// TwinCAT 3 PLC project MONETcommon
// Title: MONETcommon
// Company: IAG
// ProjectVersion: 0.5.0
// ProgramVersion: 3.1.4024.0
// libraries:
//   AstroBROT, * (BROT)
//   BROTLib, * (BROT)
//   HalfBROT, * (BROT)
//   Tc2_MC2, * (Beckhoff Automation GmbH)
//   Tc2_Standard, * (Beckhoff Automation GmbH)
//   Tc2_System, * (Beckhoff Automation GmbH)
//   Tc2_Utilities, * (Beckhoff Automation GmbH)
// project tree:
//   / E_ModeLanguage.TcDUT, FB_MonetCabinetControl.TcPOU, FB_MonetCoverControl.TcPOU, FB_MonetDiagnostics.TcPOU, FB_MonetMqttWatchdog.TcPOU, FB_MonetPendantControl.TcPOU, FB_MonetPowerMonitoring.TcPOU, FB_MonetSafetyHandling.TcPOU, F_AzimuthOffsetOnAxis.TcPOU, FB_MonetTelescopeControl.TcPOU, Global_Version.TcGVL

// ---- E_ModeLanguage.TcDUT
TYPE E_ModeLanguage :(Deutsch:=1,English:=2);


END_TYPE

// ---- Global_Version.TcGVL
{attribute 'qualified_only'}
VAR_GLOBAL CONSTANT
	// Mirrors Beckhoff's own Global_Version.stLibVersion_* pattern (see ST_LibVersion),
	// which only covers Tc2_*/Tc3_* library references, not custom ones -- until now: this
	// GVL uses Beckhoff's own naming exactly, so it merges into a consumer's Global_Version.
	// Kept in sync with <ProjectVersion> in MONETcommon.plcproj at release time.
	stLibVersion_MONETcommon : ST_LibVersion := (
		iMajor := 0,
		iMinor := 5,
		iBuild := 0,
		iRevision := 0,
		nFlags := 1,
		sVersion := '0.5.0'
	);
END_VAR

// ---- FB_MonetCabinetControl.TcPOU
FUNCTION_BLOCK FB_MonetCabinetControl
VAR_INPUT
END_VAR
VAR_OUTPUT
	bCabinetOverTemp	: BOOL;	// cabinet temperature (BT1) is critical (>60°C); not wired to any stop/park action yet, see MONETcommon#21
END_VAR
VAR
	// AT%I*/AT%Q* below are mapped directly on this FB: only one instance per PLC is
	// supported, a second instance would collide on the same physical hardware.
	inKeyLocal			AT%I*: BOOL;	//DIN3 0.2
	inButtonStart		AT%I*: BOOL;	//DIN4 0.3
	inButtonStop		AT%I*: BOOL;	//DIN5 0.4
	inButtonReset		AT%I*: BOOL;	//DIN8 0.7
	inCabinetTemp		AT%I*: INT;		//BT1	
	inKeyClearBrakes	AT%I*: BOOL;	//DIN15 1.6
	outLampPower		AT%Q*: BOOL;	//DOUT1 0.0
	outLampManual		AT%Q*: BOOL;	//DOUT2 0.1
	outLampError		AT%Q*: BOOL;	//DOUT3 0.2	
	cabinetTemp				: REAL;
	tempWarning				: SR;
	tempCritical			: SR;
	tempEvent				: FB_EventLog;
	tempCriticalEvent		: FB_EventLog;
	blinkErrorLamp			: FB_BLINK;
	blinkPowerLamp			: FB_BLINK;
	commTimer 				: TON := (PT:=T#5S);
	fbComm					: I_Comm;
END_VAR

// check temperature
cabinetTemp := INT_TO_REAL(inCabinetTemp) / 10.0;
tempWarning(SET1 := cabinetTemp > 50.0, RESET := cabinetTemp < 40.0);
tempCritical(SET1 := cabinetTemp > 60.0, RESET := cabinetTemp < 50.0);
bCabinetOverTemp := tempCritical.Q1;

// blinking lights
blinkErrorLamp(Q => outLampError);
blinkPowerLamp(Q => outLampPower);

// telemetry
commTimer(IN:=TRUE);
IF commTimer.Q THEN
	commTimer(IN:=FALSE);
	fbComm.Publish('electronics', 'base', 'MainCabinetTemperature', LREAL_TO_FMTSTR(cabinetTemp, 2, TRUE));
END_IF

// events
tempEvent(	
	Trigger 		:= tempWarning.Q1, 
	Level 			:= ADSLOG_MSGTYPE_WARN,
	FormatString 	:= 'Main cabinet temperature warning:	%s',
	OnMessage 		:= LREAL_TO_FMTSTR(cabinetTemp, 1, TRUE),
	comm			:= fbComm);
tempCriticalEvent(	
	Trigger 		:= tempCritical.Q1, 
	Level 			:= ADSLOG_MSGTYPE_ERROR,
	FormatString 	:= 'Main cabinet temperature is critical:	%s!',
	OnMessage 		:= LREAL_TO_FMTSTR(cabinetTemp, 1, TRUE),
	comm			:= fbComm);

// deprecated: kept for existing callers (MONETN, MONETS MAIN), use AreBrakesCleared instead
METHOD PUBLIC AreBreakesCleared : BOOL
VAR_INPUT
END_VAR
AreBreakesCleared := THIS^.AreBrakesCleared();
END_METHOD

METHOD PUBLIC AreBrakesCleared : BOOL
VAR_INPUT
END_VAR
AreBrakesCleared := inKeyClearBrakes;
END_METHOD

//FB_Init is always available implicitly and it is used primarily for initialization.
//The return value is not evaluated. For a specific influence, you can also declare the
//methods explicitly and provide additional code there with the standard initialization
//code. You can evaluate the return value.
METHOD FB_Init: BOOL
VAR_INPUT
    bInitRetains	: BOOL; // TRUE: the retain variables are initialized (reset warm / reset cold)
    bInCopyCode		: BOOL;  // TRUE: the instance will be copied to the copy code afterward (online change)
	comm			: I_Comm;	   
END_VAR
THIS^.fbComm := comm;
END_METHOD

METHOD PUBLIC IsResetPushed : BOOL
VAR_INPUT
END_VAR
IsResetPushed := inButtonReset;
END_METHOD

METHOD PUBLIC IsStartPushed : BOOL
VAR_INPUT
END_VAR
IsStartPushed := inButtonStart;
END_METHOD

METHOD PUBLIC IsStopPushed : BOOL
VAR_INPUT
END_VAR
IsStopPushed := NOT inButtonStop;
END_METHOD

PROPERTY KeyLocal : BOOL
GET
KeyLocal := inKeyLocal;
END_GET
END_PROPERTY

METHOD PUBLIC SetBlinkError : BOOL
VAR_INPUT
	mode	: E_Blink;
END_VAR
blinkErrorLamp.blink := mode;
END_METHOD

METHOD PUBLIC SetBlinkPower : BOOL
VAR_INPUT
	mode	: E_Blink;
END_VAR
blinkPowerLamp.blink := mode;
END_METHOD

METHOD PUBLIC SetManualLamp : BOOL
VAR_INPUT
	enable	: BOOL;
END_VAR
outLampManual := enable;
END_METHOD

END_FUNCTION_BLOCK

// ---- FB_MonetCoverControl.TcPOU
FUNCTION_BLOCK FB_MonetCoverControl IMPLEMENTS I_MirrorCovers
VAR_INPUT
	bReset				: BOOL;		// resets all drives after an error has occurred
	// M3: bOpen/bClose are also written internally (cleared on completion) and are meant
	// to be driven only via the Open()/Close() methods, not wired externally every scan
	// (consumers currently call CoverControl() with no parameters).
	bOpen				: BOOL;		// open the cover in proper order
	bClose				: BOOL;		// close the cover in proper order
	
	// telemetry interval
	fTelemetryInterval		: TIME := T#5S;	
END_VAR
VAR_OUTPUT
	bAllOpen			: BOOL;		// all covers are open
	bAllClosed			: BOOL;		// all covers are closed
	bError				: BOOL;		// any cover-driver reports an error
END_VAR
VAR
	fbComm				: I_Comm;
	tonComm 			: TON := (PT:=fTelemetryInterval);	

	// AT%I*/AT%Q* below are mapped directly on this FB: only one instance per PLC is
	// supported, a second instance would collide on the same physical hardware.
	// output signals for opening/closing covers
	OabOpenCover  AT%Q* : ARRAY[1..3] OF BOOL;	// open cover1-3 command
	OabCloseCover AT%Q* : ARRAY[1..3] OF BOOL;   // close cover1-3 command
	
	// limit switches
	IabCoverOpen	AT%I* : ARRAY[1..3] OF BOOL;	// limit coper 1 open switch
	IabCoverClosed	AT%I* : ARRAY[1..3] OF BOOL;	// limit coper 1 closed switch
	
	// status
	abCoverOpen			: ARRAY[1..3] OF BOOL;	// cover is open
	abCoverClosed		: ARRAY[1..3] OF BOOL;	// cover is closed
	abCoverError			: ARRAY[1..3] OF BOOL;	// cover has error
	afbCoverEvent			: ARRAY[1..3] OF FB_EventLog;	// cover event
	afbTimeoutEvent : ARRAY[1..3] OF FB_EventLog;	// cover has timeout

	// M3: drive timeout if a cover does not reach its target limit switch within PT;
	// TUNE PT to the actual drive on site, 60s is an untested placeholder.
	atonMoveTimeout		: ARRAY[1..3] OF TON;
	asrCoverTimeout		: ARRAY[1..3] OF SR;	// latched until bReset, see the TON note above
	abCoverTimeout		: ARRAY[1..3] OF BOOL;
	
	srErrorTrigger			: SR;	// trigger for error
	
	fbCoversOpenedEvent		: FB_EventLog; // log if covers are open
	fbCoversClosedEvent		: FB_EventLog; // log if covers are closed
	fbCoversErrorEvent		: FB_EventLog; // Event log for a generic drive error
	
	i	: UINT;
END_VAR

(*
This is the control for the two (three) telescope covers. 
The correct order for opening is 1->3->2 and for closing 2->3->1.
GVL Open and close signals are inverted
*)

// close has precedence over open
IF bClose THEN
	bOpen := FALSE;
END_IF

// do stuff for all covers
FOR i := 1 TO 3 BY 1 DO
	// limit switches are inverted
    abCoverOpen[i]   := NOT IabCoverOpen[i];
	abCoverClosed[i] := NOT IabCoverClosed[i];

	// errors occur if covers are both opened and closed
	abCoverError[i] := abCoverOpen[i] AND abCoverClosed[i];

	// M3: a cover being driven but not reaching its target switch is also an error,
	// and must stop driving the output (gated below), not just log and keep pushing.
	atonMoveTimeout[i](IN := OabOpenCover[i] OR OabCloseCover[i], PT := T#60S);
	asrCoverTimeout[i](SET1 := atonMoveTimeout[i].Q, RESET := bReset, Q1 => abCoverTimeout[i]);
	abCoverError[i] := abCoverError[i] OR abCoverTimeout[i];
END_FOR;

// close 2->3->1
OabCloseCover[2] := bClose AND NOT abCoverClosed[2] AND NOT abCoverTimeout[2];
OabCloseCover[3] := bClose AND NOT abCoverClosed[3] AND abCoverClosed[2] AND NOT abCoverTimeout[3];
OabCloseCover[1] := bClose AND NOT abCoverClosed[1] AND abCoverClosed[2] AND abCoverClosed[3] AND NOT abCoverTimeout[1];

// open 1->3->2
OabOpenCover[1] := bOpen AND NOT abCoverOpen[1] AND NOT abCoverTimeout[1];
OabOpenCover[3] := bOpen AND NOT abCoverOpen[3] AND abCoverOpen[1] AND NOT abCoverTimeout[3];
OabOpenCover[2] := bOpen AND NOT abCoverOpen[2] AND abCoverOpen[1] AND abCoverOpen[3] AND NOT abCoverTimeout[2];

// we are open, if all covers are open
bAllOpen := abCoverOpen[1] AND abCoverOpen[2] AND abCoverOpen[3];
// we are closed, if all covers are closed
bAllClosed := abCoverClosed[1] AND abCoverClosed[2] AND abCoverClosed[3];

// error indicates an axis error on any axis
srErrorTrigger(
	SET1 := abCoverError[1] OR abCoverError[2] OR abCoverError[3],
	RESET := bReset,
	Q1 => bError);

// clear reset, if no error present
IF NOT bError THEN
	bReset := FALSE;
END_IF

IF bAllClosed THEN
	bClose := FALSE;
END_IF

IF bAllOpen THEN
	bOpen := FALSE;
END_IF

fbCoversErrorEvent.OnMessage := 'Cover drive error';
IF bError THEN
	IF abCoverError[3] THEN 
		fbCoversErrorEvent.OnMessage := 'Cover 3 has a drive error.';
	END_IF
	IF abCoverError[2] THEN 
		fbCoversErrorEvent.OnMessage := 'Cover 2 has a drive error.';
	END_IF
	IF abCoverError[1] THEN 
		fbCoversErrorEvent.OnMessage := 'Cover 1 has a drive error.';
	END_IF
END_IF

// send telemetry
tonComm.PT := fTelemetryInterval;	// M3: fTelemetryInterval was only applied at init otherwise
tonComm(IN:=TRUE);
IF tonComm.Q THEN // publish new payload every second
	tonComm(IN:=FALSE);
	THIS^._SendTelemetry();	
END_IF

fbCoversErrorEvent(
	Trigger 	:= bError, 
   	Level   	:= ADSLOG_MSGTYPE_ERROR, 
	comm 		:= fbComm);

// raise an error, if both opened and closed signals are activated
// handle RoboTel differently
afbCoverEvent[1](
	Trigger   	:= abCoverOpen[1] AND abCoverClosed[1],
	Level     	:= ADSLOG_MSGTYPE_ERROR, 
	OnMessage 	:= 'Cover1: limit switch error', 
	comm	 	:= fbComm);

afbCoverEvent[2](
	Trigger   	:= abCoverOpen[2] AND abCoverClosed[2],
    Level     	:= ADSLOG_MSGTYPE_ERROR, 
	OnMessage 	:= 'Cover2: limit switch error', 
	comm      	:= fbComm);

afbCoverEvent[3](
	Trigger   	:= abCoverOpen[3] AND abCoverClosed[3],
	Level     	:= ADSLOG_MSGTYPE_ERROR, 
	OnMessage 	:= 'Cover3: limit switch error', 
	comm 	  	:= fbComm);

//trigger an event, if we encounter a timeout
afbTimeoutEvent[1](
	Trigger   	:= abCoverTimeout[1],
	Level     	:= ADSLOG_MSGTYPE_ERROR,
	OnMessage 	:= 'Cover1: Timeout',
	comm 		:= fbComm);
afbTimeoutEvent[2](
	Trigger   	:= abCoverTimeout[2],
 	Level     	:= ADSLOG_MSGTYPE_ERROR,
	OnMessage 	:= 'Cover2: Timeout',
	comm 		:= fbComm);
afbTimeoutEvent[3](
	Trigger   	:= abCoverTimeout[3],
	Level     	:= ADSLOG_MSGTYPE_ERROR,
	OnMessage 	:= 'Cover3: Timeout',
	comm 		:= fbComm);

// Log if we are opened
fbCoversOpenedEvent(
	Trigger   	:= bAllOpen,
	Level     	:= ADSLOG_MSGTYPE_WARN,
	OnMessage 	:= 'All covers are open',
	comm 		:= fbComm);
	
//log if we are closed
fbCoversClosedEvent(
	Trigger   	:= bAllClosed,
	Level     	:= ADSLOG_MSGTYPE_HINT,
	OnMessage 	:= 'All covers are closed',
	comm 		:= fbComm);

METHOD _SendTelemetry : BOOL
VAR_INPUT
END_VAR
IF bAllClosed THEN
	fbComm.Publish('telescope', 'dome', 'AUXILIARY.COVER.REALPOS', '0.0');
ELSIF bAllOpen THEN
	fbComm.Publish('telescope', 'dome', 'AUXILIARY.COVER.REALPOS', '1.0');
ELSE
	fbComm.Publish('telescope', 'dome', 'AUXILIARY.COVER.REALPOS', '0.5');
END_IF
END_METHOD

METHOD Close : BOOL
VAR_INPUT
END_VAR
bOpen := FALSE;
bClose := TRUE;
END_METHOD

PROPERTY Closed : BOOL
GET
Closed := bAllClosed;
END_GET
END_PROPERTY

PROPERTY Error : BOOL
GET
Error := bError;
END_GET
END_PROPERTY

//FB_Init is always available implicitly and it is used primarily for initialization.
//The return value is not evaluated. For a specific influence, you can also declare the
//methods explicitly and provide additional code there with the standard initialization
//code. You can evaluate the return value.
METHOD FB_Init: BOOL
VAR_INPUT
    bInitRetains	: BOOL; // TRUE: the retain variables are initialized (reset warm / reset cold)
    bInCopyCode		: BOOL;  // TRUE: the instance will be copied to the copy code afterward (online change)
	comm			: I_Comm;   
END_VAR
THIS^.fbComm := comm;
END_METHOD

METHOD Open : BOOL
VAR_INPUT
END_VAR
bOpen := TRUE;
bClose := FALSE;
END_METHOD

PROPERTY Opened : BOOL
GET
Opened := bAllOpen;
END_GET
END_PROPERTY

METHOD Reset : BOOL
VAR_INPUT
END_VAR
bReset := TRUE;
Reset := TRUE;
END_METHOD

END_FUNCTION_BLOCK

// ---- FB_MonetDiagnostics.TcPOU
// Diagnostics telemetry (measurement 'diagnostics', location 'base'): telescope interrupted/ready/busy/stopped,
// per-axis error, error ID and enable, safety error/estop/state. Each value is published when it changes, plus a full
// snapshot every tHeartbeat so a human scanning history can tell the system was actively reporting, not just silent.
// Booleans are retained by the broker (FB_Comm_MQTT_Influx.Publish). Moved unchanged from MONETS's MAIN so that
// MONET/S and MONET/N share it (IAG specs/plans/2026-09-09-extended-diagnostics-telemetry-proposal.md).
FUNCTION_BLOCK FB_MonetDiagnostics
VAR_INPUT
	fbTelescope		: REFERENCE TO FB_MonetTelescopeControl;
	fbElevation		: REFERENCE TO FB_ElevationControl;
	fbAzimuth		: REFERENCE TO FB_AzimuthControl;
	fbDerotator		: REFERENCE TO FB_DerotatorControl;
	fbFocus			: REFERENCE TO FB_FocusControl;
	fbSafety		: REFERENCE TO FB_MonetSafetyHandling;
	tHeartbeat		: TIME := T#30S;	// republish the full snapshot on this cadence even with no change
END_VAR
VAR
	fbComm					: I_Comm;
	tonHeartbeat			: TON;
	bHeartbeatTick			: BOOL;
	bLastInterrupted		: BOOL;
	bLastElevationError		: BOOL;
	bLastAzimuthError		: BOOL;
	bLastDerotatorError		: BOOL;
	bLastFocusError			: BOOL;
	bLastElevationEnabled	: BOOL;
	bLastAzimuthEnabled		: BOOL;
	bLastDerotatorEnabled	: BOOL;
	bLastSafetyError		: BOOL;
	bLastSafetyEstop		: BOOL;
	bLastSafetyState		: BOOL;
	bLastTelescopeReady		: BOOL;
	bLastTelescopeBusy		: BOOL;
	bLastTelescopeStopped	: BOOL;
END_VAR

IF NOT (__ISVALIDREF(fbTelescope) AND __ISVALIDREF(fbElevation) AND __ISVALIDREF(fbAzimuth) AND
	__ISVALIDREF(fbDerotator) AND __ISVALIDREF(fbFocus) AND __ISVALIDREF(fbSafety)) THEN
	RETURN;
END_IF

tonHeartbeat(IN := TRUE, PT := tHeartbeat);
bHeartbeatTick := tonHeartbeat.Q;
IF bHeartbeatTick THEN
	tonHeartbeat(IN := FALSE);
END_IF

IF (fbTelescope.bInterrupted <> bLastInterrupted) OR bHeartbeatTick THEN
	fbComm.Publish('diagnostics', 'base', 'Interrupted', BOOL_TO_STRING(fbTelescope.bInterrupted));
	bLastInterrupted := fbTelescope.bInterrupted;
END_IF

IF (fbElevation.bError <> bLastElevationError) OR bHeartbeatTick THEN
	fbComm.Publish('diagnostics', 'base', 'ElevationError', BOOL_TO_STRING(fbElevation.bError));
	fbComm.Publish('diagnostics', 'base', 'ElevationErrorID', UDINT_TO_STRING(fbElevation.nErrorID));
	bLastElevationError := fbElevation.bError;
END_IF
IF (fbAzimuth.bError <> bLastAzimuthError) OR bHeartbeatTick THEN
	fbComm.Publish('diagnostics', 'base', 'AzimuthError', BOOL_TO_STRING(fbAzimuth.bError));
	fbComm.Publish('diagnostics', 'base', 'AzimuthErrorID', UDINT_TO_STRING(fbAzimuth.nErrorID));
	bLastAzimuthError := fbAzimuth.bError;
END_IF
IF (fbDerotator.bError <> bLastDerotatorError) OR bHeartbeatTick THEN
	fbComm.Publish('diagnostics', 'base', 'DerotatorError', BOOL_TO_STRING(fbDerotator.bError));
	fbComm.Publish('diagnostics', 'base', 'DerotatorErrorID', UDINT_TO_STRING(fbDerotator.nErrorID));
	bLastDerotatorError := fbDerotator.bError;
END_IF
IF (fbFocus.bError <> bLastFocusError) OR bHeartbeatTick THEN
	fbComm.Publish('diagnostics', 'base', 'FocusError', BOOL_TO_STRING(fbFocus.bError));
	fbComm.Publish('diagnostics', 'base', 'FocusErrorID', UDINT_TO_STRING(fbFocus.nErrorID));
	bLastFocusError := fbFocus.bError;
END_IF

IF (fbElevation.bEnable <> bLastElevationEnabled) OR bHeartbeatTick THEN
	fbComm.Publish('diagnostics', 'base', 'ElevationEnabled', BOOL_TO_STRING(fbElevation.bEnable));
	bLastElevationEnabled := fbElevation.bEnable;
END_IF
IF (fbAzimuth.bEnable <> bLastAzimuthEnabled) OR bHeartbeatTick THEN
	fbComm.Publish('diagnostics', 'base', 'AzimuthEnabled', BOOL_TO_STRING(fbAzimuth.bEnable));
	bLastAzimuthEnabled := fbAzimuth.bEnable;
END_IF
IF (fbDerotator.bEnable <> bLastDerotatorEnabled) OR bHeartbeatTick THEN
	fbComm.Publish('diagnostics', 'base', 'DerotatorEnabled', BOOL_TO_STRING(fbDerotator.bEnable));
	bLastDerotatorEnabled := fbDerotator.bEnable;
END_IF

IF (fbSafety.error <> bLastSafetyError) OR bHeartbeatTick THEN
	fbComm.Publish('diagnostics', 'base', 'SafetyError', BOOL_TO_STRING(fbSafety.error));
	bLastSafetyError := fbSafety.error;
END_IF
IF (fbSafety.estop <> bLastSafetyEstop) OR bHeartbeatTick THEN
	fbComm.Publish('diagnostics', 'base', 'SafetyEstop', BOOL_TO_STRING(fbSafety.estop));
	bLastSafetyEstop := fbSafety.estop;
END_IF
IF (fbSafety.state <> bLastSafetyState) OR bHeartbeatTick THEN
	fbComm.Publish('diagnostics', 'base', 'SafetyState', BOOL_TO_STRING(fbSafety.state));
	bLastSafetyState := fbSafety.state;
END_IF

IF (fbTelescope.bReady <> bLastTelescopeReady) OR bHeartbeatTick THEN
	fbComm.Publish('diagnostics', 'base', 'TelescopeReady', BOOL_TO_STRING(fbTelescope.bReady));
	bLastTelescopeReady := fbTelescope.bReady;
END_IF
IF (fbTelescope.bBusy <> bLastTelescopeBusy) OR bHeartbeatTick THEN
	fbComm.Publish('diagnostics', 'base', 'TelescopeBusy', BOOL_TO_STRING(fbTelescope.bBusy));
	bLastTelescopeBusy := fbTelescope.bBusy;
END_IF
IF (fbTelescope.bStopped <> bLastTelescopeStopped) OR bHeartbeatTick THEN
	fbComm.Publish('diagnostics', 'base', 'TelescopeStopped', BOOL_TO_STRING(fbTelescope.bStopped));
	bLastTelescopeStopped := fbTelescope.bStopped;
END_IF

METHOD FB_Init: BOOL
VAR_INPUT
    bInitRetains	: BOOL; // TRUE: the retain variables are initialized (reset warm / reset cold)
    bInCopyCode		: BOOL;  // TRUE: the instance will be copied to the copy code afterward (online change)
	comm			: I_Comm;
END_VAR
THIS^.fbComm := comm;
END_METHOD

END_FUNCTION_BLOCK

// ---- FB_MonetTelescopeControl.TcPOU
FUNCTION_BLOCK FB_MonetTelescopeControl EXTENDS FB_AltAzTelescopeControl IMPLEMENTS I_AltAzTelescope
VAR_INPUT
	fbFocus				: I_Focus;
	fbCovers			: I_MirrorCovers;
	fbBrake				: I_Brake;	
	fbHydraulics   		: I_Hydraulics;
	fbElevation			: REFERENCE TO FB_ElevationControl;
	fbAzimuth			: REFERENCE TO FB_AzimuthControl;
	fbDerotator			: REFERENCE TO FB_DerotatorControl;

	fbPointing			: REFERENCE TO FB_PointingModelForward;
	fbPointingInverse	: REFERENCE TO FB_PointingModelInversion;

	bBrakeClearing		: BOOL	:= TRUE;

	// M6: applied to every commanded elevation move (Goto/Home/Park/PowerOn/Slew, not
	// the computed tracking rate), NOT just _HomeTelescope despite the old name.
	// 5.0 deg/s confirmed correct on-site for MONETS; 10.0 was too fast.
	fElevationMoveVelocity : LREAL := 5.0;
END_VAR
VAR_OUTPUT
	fDerotatorSign		: LREAL := 1.0;	// derotator
	
	fElevationPointingOffset : LREAL;
	fAzimuthPointingOffset : LREAL;
	fElevationPointingOffset2 : LREAL;
	fAzimuthPointingOffset2 : LREAL;
	
	fRightAscensionCurrentSky: LREAL;
	fDeclinationCurrentSky: LREAL;

	fDerotatorVelocity	: LREAL;	// rotational velocity of the derotator
	fElevationVelocity	: LREAL;	// rotational velocity of the elevation
	fAzimuthVelocity	: LREAL;	// rotational velocity of the elevation
END_VAR
VAR
	// M1: internal (non-axis) errors from the Goto/Home/Slew state machines, latched
	// until bReset since bError/nErrorID are otherwise recomputed from the axes every
	// scan and would silently wipe these within the same cycle they're set in.
	bSoftwareError		: BOOL;
	nSoftwareErrorID	: UINT;
	SoftwareErrorEvent	: FB_EventLog;

	// #26 / ADR 0001 option 1: auto-clear a latched bInterrupted if nothing has been
	// requested for a while, since the normal arbitration path can never do it on its
	// own (bReady needs the axes enabled, axis enable needs bInterrupted already clear).
	// Visible, not silent: logged and counted, not just quietly cleared.
	bInterruptedIdle			: BOOL;
	tonInterruptedAutoClear		: TON;
	InterruptedAutoClearEvent	: FB_EventLog;
END_VAR
VAR PERSISTENT
	nInterruptedAutoClearCount	: UDINT;	// how many times auto-clear has fired, ever
END_VAR

// revert fDut1 (set via the Dut1 property, e.g. from an external time bridge over MQTT) to its
// safe 0.0 default if nothing fresh arrives for a while, instead of serving an arbitrarily
// stale UT1-UTC correction forever. FB_AltAzTelescopeControl's own body is never called (this FB
// doesn't call SUPER^() in its main body), so this has to live here rather than up there.
tonDut1Stale(IN := NOT bDut1Received, PT := T#10M);
bDut1Received := FALSE;
IF tonDut1Stale.Q THEN
	fDut1 := 0.0;
END_IF

// get the system time; fJd only follows the clock while the clock is valid (synced, see FB_AstroClock)
fbTime();
IF fbTime.bValid THEN
	fJd := DateTime2JD(fbTime.time_RTCEX2);
END_IF
fLst := CT2LST(telescopeConfig.longitude, fJd);

// without a trustworthy time nothing may be pointed or tracked: refuse through the normal stop path
IF NOT fbTime.bValid AND (bGoto OR bSlew OR bTrack) THEN
	bStop := TRUE;
END_IF

// set reset state either by hardware (key pressed) or by software (set by e.g. tcs)
rtrigReset(CLK := bReset);

IF bReset THEN
	bHorizonError := FALSE; // if reset, the bHorizonError can be switched off
	bSoftwareError := FALSE;
	
	// reset the stages of all statemachine methods
	bInterrupted := TRUE; 
	_HomeTelescope();
	_GotoTelescope();
	_SlewTelescope();
	_ParkTelescope();
	bInterrupted := FALSE;
END_IF

// get error ID, reset if bReset command is set
IF fbAzimuth.Error THEN
	nErrorID := fbAzimuth.nErrorID;
	IF bReset THEN
		fbAzimuth.Reset();
	END_IF
ELSIF fbElevation.bError THEN
	nErrorID := fbElevation.nErrorID;
	IF bReset THEN
		fbElevation.Reset();
	END_IF
ELSIF fbDerotator.bError THEN
	nErrorID := fbDerotator.nErrorID;
	IF bReset THEN
		fbDerotator.Reset();
	END_IF	
ELSIF fbFocus.Error THEN
	nErrorID := fbFocus.ErrorID;
	IF bReset THEN
		fbFocus.Reset();
	END_IF
ELSIF bSoftwareError THEN
	nErrorID := nSoftwareErrorID;
END_IF

// fSlewTime
fSlewTime :=  MAX(MAX(fbElevation.fSlewTime, fbAzimuth.fSlewTime), fbDerotator.fSlewTime);

bError := fbElevation.Error OR
		 fbAzimuth.bError OR
		 fbFocus.Error OR
		 fbDerotator.bError OR
		 bSoftwareError;
			
IF bError THEN
	bTrack := 	FALSE;
	bGoto := 	FALSE;
	bSlew := 	FALSE;
	fbElevation.Enable := FALSE;
	fbAzimuth.Enable := FALSE;
	fbDerotator.Enable := FALSE;
ELSE
	nErrorID := 0;
END_IF

IF fbElevation.bError THEN
	fbElevation.Enable := FALSE;
	fbAzimuth.Enable := FALSE;
	fbDerotator.Enable := FALSE;
	fbBrake.CloseBrake();
END_IF

eq2hor(
	ra := fRightAscension,
	dec := fDeclination,
	lon := telescopeConfig.longitude,
	lat := telescopeConfig.latitude,
	altitude := telescopeConfig.altitude,
	JD := fJd + fTimeOffset,
	dut1 := fDut1,
	refract_to_observed := TRUE,
	// refract := FALSE,
	alt => fElevationCalc,
	az => fAzimuthCalc,
	ha => fHourAngleCalc);

// apply pointing model
fbPointing(
	fAzimuth			:= fAzimuthCalc,
	fElevation			:= fElevationCalc,
	fAzimuthOffset		=> fAzimuthPointingOffset,
	fElevationOffset	=> fElevationPointingOffset
);
fElevationCalc := fElevationCalc + fElevationPointingOffset + fElevationOffset;
// F_AzimuthOffsetOnAxis: fAzimuthOffset / COS(elevation), bounded near the zenith (BROTLib#27)
fAzimuthCalc := fAzimuthCalc + fAzimuthPointingOffset + F_AzimuthOffsetOnAxis(fAzimuthOffset, fElevationCalc);

// calculate derotator position 
fDerotatorCalc := F_DerotatorPosition2(fAzimuthCalc, fElevationCalc, telescopeConfig.latitude, fDerotatorSign)  + fDerotatorOffset;

// calculate velocities
fDerotatorVelocity := F_Derotatorvelocity(fAzimuthCalc, fElevationCalc, telescopeConfig.latitude, fDerotatorSign);
fElevationVelocity := F_Elevationvelocity(fAzimuthCalc, telescopeConfig.latitude);
fAzimuthVelocity := F_Azimuthvelocity(fElevationCalc, fAzimuthCalc, telescopeConfig.latitude);

IF (fAzimuthCalc > 310.0 AND fAzimuthVelocity > 0.0) OR (fAzimuthCalc > 440.0) THEN
	fAzimuthCalc := fAzimuthCalc - 360.0;
ELSIF (fAzimuthCalc < 80.0 AND fAzimuthVelocity < 0.0) OR (fAzimuthCalc < -50.0) THEN
	fAzimuthCalc := fAzimuthCalc + 360.0;
END_IF

IF (fDerotatorCalc > 290.0 AND fDerotatorVelocity > 0.0) OR (fDerotatorCalc > 380.0) THEN
	fDerotatorCalc := fDerotatorCalc - 360.0;
ELSIF (fDerotatorCalc < 20.0 AND fDerotatorVelocity < 0.0) OR (fDerotatorCalc < -70.0) THEN
	fDerotatorCalc := fDerotatorCalc + 360.0;
END_IF

// get current coordinates	
fAzimuthCurrent := fbAzimuth.fActualPosition;
fElevationCurrent := fbElevation.fActualPosition;
fDerotatorCurrent := fbDerotator.fActualPosition;

// apply inverse pointing model
fbPointingInverse(
	fAzimuth			:= fAzimuthCurrent,
	fElevation			:= fElevationCurrent,
	fAzimuthOffset  	=> fAzimuthPointingOffset2,
	fElevationOffset	=> fElevationPointingOffset2
);
fAzimuthCurrentSky := fAzimuthCurrent - fAzimuthPointingOffset2;
fElevationCurrentSky := fElevationCurrent - fElevationPointingOffset2;

// add offsets
//fElevationCurrent := fElevationCurrentSky - fElevationOffset;
//fAzimuthCurrent := fAzimuthCurrentSky - fAzimuthOffset / COS(fElevationCalc * d2r);

// calculate equatorial coordinates
hor2eq(alt := fElevationCurrentSky - fElevationOffset,
		az := fAzimuthCurrentSky - F_AzimuthOffsetOnAxis(fAzimuthOffset, fElevationCurrent),	// M7: was fElevationCalc
		jd := fJd,
		dut1 := fDut1,
		lat := telescopeConfig.latitude,
		lon := telescopeConfig.longitude,
		altitude := telescopeConfig.altitude,
		alt_is_observed := TRUE,
		// refract := FALSE,
		ra => fRightAscensionCurrent,
		dec => fDeclinationCurrent,
		ha => fHourAngleCurrent);	// M13: was never assigned, HA_ICRS telemetry was stuck at 0.0
hor2eq(alt := fElevationCurrentSky,
		az := fAzimuthCurrentSky,
		jd := fJd,
		dut1 := fDut1,
		lat := telescopeConfig.latitude,
		lon := telescopeConfig.longitude,
		altitude := telescopeConfig.altitude,
		alt_is_observed := TRUE,
		ra => fRightAscensionCurrentSky,
		dec => fDeclinationCurrentSky);
	
// If the Telescope dips under the fHorizon (e.g. while tracking, stop and gohome)
IF fbElevation.Calibrated AND fElevationCurrent < (fHorizon+0.2) THEN
	IF NOT bStopped AND NOT bGoHome THEN
		bStop := TRUE;
	ELSE
		bGoHome := TRUE;
	END_IF
END_IF
		
tpPowerOnWarning(IN := bPower OR (NOT fbElevation.bEnable AND fbBrake.BrakeOpen), PT := T#250MS);

tonPowerTimeout(IN := TCS_command = E_TCSCommand.no_command AND NOT bIsParked, PT := T#12H);
tonCommandTimeout();
IF tonPowerTimeout.Q AND NOT bIsParked THEN
	bPark := TRUE;
END_IF
		
// #26 / ADR 0001 option 1: bInterrupted otherwise cannot clear itself once latched with
// nothing pending (see specs/design/telescopecontrol-command-arbitration.md); auto-clear
// after a few seconds of true idle (no error, nothing requested), logged and counted so
// it's visible rather than a silent recovery. TUNE PT if this fires too eagerly/late on
// site.
bInterruptedIdle := bInterrupted AND NOT bError AND
	NOT (bPower OR bPark OR bGoHome OR bGoto OR bSlew OR bTrack);
tonInterruptedAutoClear(IN := bInterruptedIdle, PT := T#5S);
IF tonInterruptedAutoClear.Q THEN
	bInterrupted := FALSE;
	nInterruptedAutoClearCount := nInterruptedAutoClearCount + 1;
END_IF
InterruptedAutoClearEvent(
	Trigger 		:= tonInterruptedAutoClear.Q,
	Level 			:= ADSLOG_MSGTYPE_WARN,
	FormatString 	:= 'bInterrupted auto-cleared after idle timeout (count: %s)',
	OnMessage 		:= UDINT_TO_STRING(nInterruptedAutoClearCount),
	Comm 			:= fbComm);

// set TCS_command according to state variables ordered by precedence
// Stop outranks everything, including a running power-on
IF bStop THEN
	bTrack := FALSE;
	
	// If the stop is during a power-on or a movement, reset the stage of the movement first
	IF bPower THEN
		bPower := FALSE;
		_PowerOn();
	END_IF
	IF bPark THEN
		bPark := FALSE;
		_ParkTelescope();
	ELSIF bGoto THEN
		bGoto := FALSE;
		_GotoTelescope();
	ELSIF bSlew THEN
		bSlew := FALSE;
		_SlewTelescope();
	ELSIF bGoHome THEN
		bGoHome := FALSE;
		_HomeTelescope();
	END_IF
	TCS_command := E_TCSCommand.stop;
	
ELSIF bPower THEN
	TCS_command := E_TCSCommand.poweron;
	
ELSIF bPark THEN
	bTrack := FALSE;
	// M2: emergency park bypasses the bReady/bBusy gating below entirely, since bReady
	// requires NOT bError and would otherwise make park unreachable during an error.
	IF bError THEN
		bInterrupted := FALSE;
		TCS_command := E_TCSCommand.park;
	// If lower presedence commands are ongoing, let them know they are interupted
	ELSIF bGoto OR bSlew OR bGoHome THEN
		bGoHome := FALSE;
		bGoto := FALSE;
		bSlew := FALSE;
		bInterrupted := TRUE;
		_HomeTelescope();
		_GotoTelescope();
		_SlewTelescope();

	ELSE
		IF bReady AND NOT bBusy THEN
			bInterrupted := FALSE;
			TCS_command := E_TCSCommand.park;
		END_IF
	END_IF
	
ELSIF bGoHome THEN
	bTrack := FALSE;
	// If lower presedence commands are ongoing, let them know they are interupted
	IF bGoto OR bSlew THEN
		bGoto := FALSE;
		bSlew := FALSE;
		bInterrupted := TRUE;
		_GotoTelescope();
		_SlewTelescope();
		
	ELSE
		IF bReady AND NOT bBusy AND bStopped THEN
			bInterrupted := FALSE;
			TCS_command := E_TCSCommand.gohome;
		END_IF
	END_IF
	
	
ELSIF bGoto THEN
	bTrack := FALSE;
	// If lower presedence commands are ongoing, let them know they are interupted
	IF bSlew THEN
		bSlew := FALSE;
		bInterrupted := TRUE;
		_SlewTelescope();
	ELSE
		IF bReady AND NOT bBusy THEN
			bInterrupted := FALSE;
			TCS_command := E_TCSCommand.goto;
		END_IF
	END_IF
		
ELSIF bSlew THEN
	bTrack := FALSE;
	IF bReady AND NOT bBusy THEN
		TCS_command := E_TCSCommand.slew;
	END_IF
	
ELSIF bTrack THEN
	IF bReady AND NOT bBusy THEN
		TCS_command := E_TCSCommand.track;
	END_IF
	
ELSE
	TCS_command := E_TCSCommand.no_command;
	fbElevation.bMoveAxis := FALSE;
	fbAzimuth.bMoveAxis := FALSE;
	fbDerotator.bMoveAxis := FALSE;
	fbElevation.bTracking := FALSE;
	fbAzimuth.bTracking := FALSE;
	fbDerotator.bTracking := FALSE;
END_IF

IF TCS_command = E_TCSCommand.poweron THEN
	_PowerOn();
	tonCommandTimeout(IN := TCS_command = E_TCSCommand.poweron, PT := T#12H);
	TCSCTOEvent.OnMessage := 'POWER';
ELSIF TCS_command = E_TCSCommand.stop THEN
	_StopTelescope();
	tonCommandTimeout(IN := TCS_command = E_TCSCommand.stop, PT := T#2S);
	TCSCTOEvent.OnMessage := 'STOP';
ELSIF TCS_command = E_TCSCommand.park THEN
	_ParkTelescope();
	tonCommandTimeout(IN := TCS_command = E_TCSCommand.park, PT := T#2M);
	TCSCTOEvent.OnMessage := 'PARK';
ELSIF TCS_command = E_TCSCommand.gohome THEN
	_HomeTelescope();
	tonCommandTimeout(IN := TCS_command = E_TCSCommand.gohome, PT := T#2M);
	TCSCTOEvent.OnMessage := 'GOHOME';
ELSIF TCS_command = E_TCSCommand.goto THEN
	_GotoTelescope();
	tonCommandTimeout(IN := TCS_command = E_TCSCommand.goto, PT := T#2M);
	TCSCTOEvent.OnMessage := 'GOTO';
ELSIF TCS_command = E_TCSCommand.slew THEN
	_SlewTelescope();
	tonCommandTimeout(IN := TCS_command = E_TCSCommand.slew, PT := T#2M);
	TCSCTOEvent.OnMessage := 'SLEW';
ELSIF TCS_command = E_TCSCommand.track THEN
	_TrackTelescope();
	tonCommandTimeout(IN := TCS_command = E_TCSCommand.track, PT := T#12H);
	TCSCTOEvent.OnMessage := 'TRACK';
ELSE
	// disable command timeout
	tonCommandTimeout(IN := FALSE);
	TCSCTOEvent.OnMessage := 'NOCOMMAND';
END_IF
 
bSlewing := NOT bTracking AND (fbElevation.fbAxis.InMotion OR fbElevation.fbAxis.InRamp OR
			fbAzimuth.fbAxis.InMotion OR fbAzimuth.fbAxis.InRamp OR
			fbDerotator.fbAxis.InMotion OR fbDerotator.fbAxis.InRamp);

// signal must be stable for 5500MS
tonTrackingDelay(in := fbElevation.fbAxis.isTracking AND 
			fbAzimuth.fbAxis.isTracking AND
			fbDerotator.fbAxis.isTracking,PT :=T#5500MS, Q => bTracking);
			
bStopped :=  (NOT fbElevation.bEnable OR fbElevation.fbAxis.StandStill) AND 
			(NOT fbAzimuth.bEnable OR fbAzimuth.fbAxis.StandStill) AND
			(NOT fbDerotator.bEnable OR fbDerotator.fbAxis.StandStill);
			
bHomed := fbElevation.Calibrated AND
			fbAzimuth.Calibrated AND
			fbFocus.Calibrated AND
			fbDerotator.Calibrated;
			
bReady := bHomed AND 
	fbCovers.Opened AND 
	fbElevation.bEnable AND
	fbAzimuth.bEnable AND
	fbDerotator.bEnable AND fbBrake.BrakeOpen AND 
    NOT bError;

bBusy := fbElevation.fbAxis.Busy OR
		fbAzimuth.fbAxis.Busy OR
		fbDerotator.fbAxis.Busy OR
		fbFocus.Busy;

(* STATUS STATES*)
//fReadyState (see also _PowerOn and _ParkTelescope calls above)
IF bError THEN
	fReadyState := -1.0;
ELSIF bPower THEN
	fReadyState := 0.7;
ELSIF bIsParked THEN
	fReadyState := 0.0;
ELSIF bPark THEN
	fReadyState := 0.3;
ELSIF bReady THEN
	fReadyState := 1.0;	
ELSE
	fReadyState := -2.0;	
END_IF

//MotionState
IF bStopped THEN
	nMotionState := 0;
ELSIF bSlewing OR bBusy THEN
	nMotionState := 1;
ELSIF bTracking THEN
	nMotionState := 8;
END_IF

// unset the STOP command if telescope is already stopped
IF bStopped THEN
	bStop := FALSE;
END_IF
	
IF NOT bError THEN
	bReset := FALSE;
END_IF

IF bEstopTriggered THEN
	fbElevation.Enable := FALSE;
	fbAzimuth.Enable := FALSE;
	fbDerotator.Enable := FALSE;
END_IF

// send telemetry
IF bSlewing OR bTrack OR bTracking THEN
	tonMQTTTimer.PT := T#500MS; // M13: was "every second", actually twice a second while moving
ELSE
	tonMQTTTimer.PT := T#1000MS; // M13: was "every five seconds", actually every second otherwise
END_IF
tonMQTTTimer(IN:=TRUE);
IF tonMQTTTimer.Q THEN
	tonMQTTTimer(IN:=FALSE);
	_SendTelemetry();
END_IF


(* Event function blocks start here. *)
TCSpowerEvent(	Trigger := bPowerFailure, 
				Level := ADSLOG_MSGTYPE_ERROR,
				FormatString := 'power %s',
				//OnMessage := 'Failure',
				OffMessage := 'OK', 
				Comm := fbComm);

TCSgohomeEvent(	Trigger := bGoHome, 
				Level := ADSLOG_MSGTYPE_HINT,
				FormatString := 'GOHOME %s',
				OnMessage := 'commencing',
				OffMEssage := 'completed', 
				Comm := fbComm);
TCSparkEvent(	Trigger := bPark, 
				Level := ADSLOG_MSGTYPE_HINT,
				FormatString := 'PARK %s',
				OnMessage := 'commencing',
				OffMEssage := 'completed', 
				Comm := fbComm);
TCSgotoEvent(	Trigger := bGoto, 
				Level := ADSLOG_MSGTYPE_HINT,
				FormatString := 'GOTO %s',
				OnMessage := 'commencing',
				OffMEssage := 'completed', 
				Comm := fbComm);
TCStrackEvent(	Trigger := bTrack, 
				Level := ADSLOG_MSGTYPE_HINT,
				FormatString := 'TRACK %s',
				OnMessage := 'commencing',
				OffMEssage := 'completed', 
				Comm := fbComm);
TCSstopEvent(	Trigger := bStop, 
				Level := ADSLOG_MSGTYPE_WARN,
				FormatString := 'STOP %s',
				OnMessage := 'commencing',
				OffMEssage := 'completed',
				OffLevel := ADSLOG_MSGTYPE_HINT, 
				Comm := fbComm);
TCStargetHorizonEvent(	Trigger := fElevationCalc<fHorizon,
				Level := ADSLOG_MSGTYPE_WARN,
				FormatString := '%s',
				OnMessage := 'Target below safe horizon',
				OffMEssage := '', 
				Comm := fbComm);
TCSreadyEvent(	Trigger := bPower AND bReady, 
				Level := ADSLOG_MSGTYPE_HINT,
				FormatString := '%s',
				OnMessage := 'STELLA1 startup finished', 
				Comm := fbComm);
TCSCTOEvent(	Trigger := tonCommandTimeout.Q,
				Level := ADSLOG_MSGTYPE_WARN,
				FormatString := 'A timeout occurred during %s command!',
				OnMessage := 'NOCOMMAND',
				Comm := fbComm);
SoftwareErrorEvent(	Trigger := bSoftwareError,
				Level := ADSLOG_MSGTYPE_ERROR,
				FormatString := 'Internal command error, ID: %s',
				OnMessage := UINT_TO_STRING(nSoftwareErrorID),
				OffMessage := 'cleared',
				OffLevel := ADSLOG_MSGTYPE_HINT,
				Comm := fbComm);

METHOD PRIVATE _GotoTelescope : USINT
VAR_INPUT
END_VAR
VAR
	GoToEvent		: FB_Eventlog;
	commandTimeout	: TON;
END_VAR
VAR_STAT
	nStage			: USINT := 0;
	nLastStage		: USINT := 101;
END_VAR
_GotoTelescope := nStage;
commandTimeout(IN := nStage < 100, PT := T#600S);
IF commandTimeout.Q THEN
	bError := TRUE;
	nErrorID := 16#10;
	bSoftwareError := TRUE;
	nSoftwareErrorID := 16#10;
	bGoto := FALSE;
	nStage := 0;
	RETURN;
END_IF

IF fElevationCalc<2.0 THEN
	bError := TRUE;
	nErrorID := 16#15;
	bSoftwareError := TRUE;
	nSoftwareErrorID := 16#15;
	bGoto := FALSE;
	nStage := 0;
	RETURN;
END_IF

// M7: near zenith COS(elevation) -> 0, so any nonzero fAzimuthOffset blows up into a
// huge azimuth (see the offset divisions elsewhere in this FB). 89.5 matches the
// existing tracking cutoff (_TrackTelescope: fElevationCurrent > 89.5).
IF fElevationCalc>89.5 THEN
	bError := TRUE;
	nErrorID := 16#16;
	bSoftwareError := TRUE;
	nSoftwareErrorID := 16#16;
	bGoto := FALSE;
	nStage := 0;
	RETURN;
END_IF

IF bReset OR bError OR bInterrupted THEN
	nStage := 0;
	RETURN;
END_IF

CASE nStage OF
	0:	
		IF bReady AND NOT bBusy THEN
			nStage := 10;
		END_IF
	10:
		IF fbElevation.Tracking = TRUE OR fbAzimuth.Tracking = TRUE OR fbDerotator.Tracking = TRUE THEN
			fbElevation.Tracking := FALSE;
			fbAzimuth.Tracking := FALSE;
			fbDerotator.Tracking := FALSE;
		ELSE
			nStage := 25;
		END_IF				
	25:	
		fbElevation.Position := fElevationCalc;
		fbAzimuth.Position := fAzimuthCalc;
		fbDerotator.Position := fDerotatorCalc;
		fbDerotator.Velocity := 10.0;
		fbElevation.Velocity := fElevationMoveVelocity;
		fbAzimuth.Velocity := 10.0;
		
		fbElevation.MoveAxis := TRUE;
		fbAzimuth.MoveAxis := TRUE;
		fbDerotator.MoveAxis := TRUE;
		IF fbElevation.Busy AND
			fbAzimuth.Busy AND
			fbDerotator.Busy THEN
				nStage := 50;
		END_IF
	50:
		IF NOT fbElevation.Busy AND fbElevation.MoveDone THEN
			fbElevation.MoveAxis := FALSE;
		END_IF
		IF NOT fbAzimuth.Busy AND fbAzimuth.MoveDone THEN
			fbAzimuth.MoveAxis := FALSE;
		END_IF
		IF NOT fbDerotator.Busy AND fbDerotator.MoveDone THEN
			fbDerotator.MoveAxis := FALSE;
		END_IF
		IF NOT fbElevation.MoveAxis AND 
           NOT fbAzimuth.MoveAxis AND 
		   NOT fbDerotator.MoveAxis THEN
		   nStage := 75;
		END_IF
	75:
		IF NOT bSlewing AND bStopped THEN // all axis standstill
			nStage := 100;
		END_IF
	100:
		fbElevation.MoveAxis := FALSE;
		fbAzimuth.MoveAxis := FALSE;
		fbDerotator.MoveAxis := FALSE;
		fAzimuth := fAzimuthCalc;
		fElevation := fElevationCalc;
		bGoto := FALSE;
		// enable automatic tracking
		bTrack := bAutoTrack;
		nStage := 0;
END_CASE
GoToEvent(Trigger := nStage > nLastStage, FormatString := 'GoTo progress: %s', OnMessage := USINT_TO_STRING(nStage), comm := fbComm);
nLastStage := nStage;
END_METHOD

METHOD PRIVATE _HomeTelescope : BOOL
VAR_INPUT
END_VAR
VAR
    HomeEvent        : FB_Eventlog;
    commandTimeout    : TON;
END_VAR
// reset/interrupt aborts the homing without moving anything, like the other stage methods
IF bReset OR bError OR bInterrupted THEN
    commandTimeout(IN := FALSE);
    RETURN;
END_IF

commandTimeout(IN := NOT _HomeTelescope, PT := T#600S);
IF commandTimeout.Q THEN
    bError := TRUE;
    nErrorID := 16#30;
    bSoftwareError := TRUE;
    nSoftwareErrorID := 16#30;
    _HomeTelescope :=TRUE;
END_IF

// only move while a home command is active (Stop/Park/Reset call this with bGoHome cleared to abort it)
IF bGoHome AND bReady AND bStopped AND NOT bBusy AND NOT bTracking THEN
    fbElevation.Velocity := fElevationMoveVelocity;
    fbElevation.Position := telescopeConfig.elevationHome;
    fbElevation.MoveAxis := TRUE;
    fbAzimuth.Velocity := 10.0;
    fbAzimuth.Position := telescopeConfig.azimuthHome;
    fbAzimuth.MoveAxis := TRUE;
    fbDerotator.Velocity := 10.0;
    fbDerotator.Position := telescopeConfig.derotatorHome;
    fbDerotator.MoveAxis := TRUE;    
END_IF

IF fbElevation.MoveDone AND 
    fbAzimuth.MoveDone AND 
    fbDerotator.MoveDone THEN
    bGoHome := FALSE;
    fElevation := fElevationCurrent;
    fAzimuth := fAzimuthCurrent;
    _HomeTelescope := TRUE;
ELSE
    _HomeTelescope := FALSE;
END_IF

HomeEvent(Trigger := _HomeTelescope, 
            Level := ADSLOG_MSGTYPE_HINT,
            FormatString := '%s',
            OnMessage := 'Telescope is homed.', comm := fbComm);
END_METHOD

METHOD PRIVATE _ParkTelescope : USINT
VAR_INPUT
END_VAR
VAR
	ParkEvent	: FB_Eventlog;
	rtrigError	: R_TRIG;	// M2: reset the stage only on the rising edge of bError, not every scan
END_VAR
VAR_STAT
	nStage		: USINT := 0;
	nLastStage	: USINT := 101;
END_VAR
_ParkTelescope := nStage;
IF bReset OR bStop OR bInterrupted THEN
	nStage := 0;
	RETURN;
END_IF
// M2: bError does NOT return early here, unlike the other state machines: stage 0's
// "emergency park" branch below is the safe-state response to bError and must run.
// Only force the stage back to 0 on the rising edge, so the emergency branch can still
// progress through its own stages (80 -> 100) on later scans while bError stays TRUE.
rtrigError(CLK := bError);
IF rtrigError.Q THEN
	nStage := 0;
END_IF
IF bIsParked THEN
	nStage := 100;
END_IF
CASE nStage OF
	0: 
		bGoHome := 	FALSE;
		bTrack := 	FALSE;
		bGoto := 	FALSE;
		bSlew := 	FALSE;
		fbFocus.Position := telescopeConfig.focusPark;
		IF bError THEN // emergency park
			fbBrake.CloseBrake();
			fbElevation.Enable := FALSE;
			fbAzimuth.Enable := FALSE;
			fbDerotator.Enable := FALSE;	
			fbCovers.Close();	
			nStage := 80;
		ELSE
			nStage := 10;
		END_IF
	10:
		IF fbElevation.Tracking = TRUE OR fbAzimuth.Tracking = TRUE OR fbDerotator.Tracking = TRUE THEN
			fbElevation.Tracking := FALSE;
			fbAzimuth.Tracking := FALSE;
			fbDerotator.Tracking := FALSE;
		ELSE
			nStage := 20;
		END_IF		
	20:
		fbElevation.Position := telescopeConfig.elevationPark;
		fbElevation.Velocity := fElevationMoveVelocity;
		fbElevation.MoveAxis := TRUE;
		fbAzimuth.Position := telescopeConfig.azimuthPark;
		fbAzimuth.Velocity := 10;
		fbAzimuth.MoveAxis := TRUE;
		fbDerotator.Position := telescopeConfig.derotatorPark;
		fbDerotator.Velocity := 10.0;
		fbDerotator.MoveAxis := TRUE;
		IF fbElevation.Busy AND
			fbAzimuth.Busy AND
			fbDerotator.Busy THEN
				nStage := 40;
		END_IF
	40:
		IF fbElevation.MoveDone THEN
			fbElevation.MoveAxis := FALSE;
		END_IF
		IF fbAzimuth.MoveDone THEN
			fbAzimuth.MoveAxis := FALSE;
		END_IF
		IF fbDerotator.MoveDone THEN
			fbDerotator.MoveAxis := FALSE;
		END_IF
		IF NOT bSlewing THEN // all axis standstill
			nStage := 60;
		END_IF
	60:
		IF NOT fbElevation.Enable AND NOT fbAzimuth.Enable AND NOT fbDerotator.Enable THEN
			nStage := 80;
		END_IF

		IF bStopped THEN
			fbElevation.Enable := FALSE;
			fbAzimuth.Enable := FALSE;
			fbDerotator.Enable := FALSE;
		END_IF
		
		fbElevation.bMoveAxis := FALSE;
		fbAzimuth.bMoveAxis := FALSE;
		fbDerotator.bMoveAxis := FALSE;
	80:
		IF fbElevation.Enable OR fbAzimuth.Enable OR fbDerotator.Enable THEN
			nStage := 60;
		END_IF
		IF NOT fbBrake.BrakeOpen THEN
			fbCovers.Close();
			fbHydraulics.Enable := FALSE;
		END_IF
		IF fbCovers.Closed THEN
			nStage := 100;
		END_IF
	100:
			bIsParked := TRUE;
			bPark := FALSE;
			_ParkTelescope := 100;
			nStage := 0;	
END_CASE
ParkEvent(Trigger := nStage > nLastStage, FormatString := 'Parking progress: %s', OnMessage := USINT_TO_STRING(nStage), comm := fbComm);
nLastStage := nStage;
END_METHOD

METHOD PRIVATE _PowerOn : BOOL
VAR_INPUT
END_VAR
VAR_STAT
	nStage		: USINT := 0;
	nLastStage	: USINT := 101;
END_VAR
IF NOT bBrakeClearing THEN
	bPowerFailure := TRUE;
	TCSpowerEvent.OnMessage := 'failure: brake clearing not set';
	bPower := FALSE;
ELSIF bError THEN
	bPowerFailure := TRUE;
	TCSpowerEvent.OnMessage := 'Generic error during power on occurred.';
	bPower := FALSE;
ELSE
	bPowerFailure := FALSE;		
END_IF

IF bReset OR bError OR bStop OR bInterrupted THEN
	nStage := 0;
	// abort without leaving the last written axis commands set
	fbElevation.MoveAxis := FALSE;
	fbElevation.HomeAxis := FALSE;
	fbAzimuth.MoveAxis := FALSE;
	fbAzimuth.HomeAxis := FALSE;
	fbDerotator.MoveAxis := FALSE;
	fbDerotator.HomeAxis := FALSE;
	fbFocus.HomeAxis := FALSE;
	RETURN;
END_IF

CASE nStage OF
	0:
		_PowerOn := FALSE;
		// COVER MUST BE OPENED FOR A SUCCESSFUL WAKE & SHAKE COMMAND!
		// unconditional by design: does not consult bCoverAutoOpen (see CoverAutoOpen.Set)
		fbCovers.Open();
		IF bMainReady AND fbCovers.Opened THEN
			nStage := 10;
		END_IF
		
	10:
		fbElevation.Enable := TRUE;
		fbAzimuth.Enable := TRUE;
		fbDerotator.Enable := TRUE;
		
		IF fbElevation.Ready AND NOT fbElevation.Calibrated THEN
			fbElevation.HomeAxis := TRUE;
		END_IF
		
		IF fbAzimuth.Ready AND NOT fbAzimuth.Calibrated THEN
			fbAzimuth.HomeAxis := TRUE;
		END_IF
		
		// enable derotator
		IF fbElevation.Ready THEN
			fbDerotator.HomeAxis := fbDerotator.Ready AND NOT fbDerotator.Calibrated;
		END_IF
		
		// start calibration of focus after elevation has been calibrated
		// this avoids imbalance by the M2 mirror on the elvation during its calibration
		IF fbElevation.Calibrated AND NOT fbFocus.Calibrated THEN
			fbFocus.Enable := TRUE;
			fbFocus.HomeAxis := TRUE;
		END_IF
	
		IF fbCovers.Opened AND fbElevation.Calibrated AND fbAzimuth.Calibrated AND fbDerotator.Calibrated AND fbFocus.Calibrated AND
			bReady AND bStopped AND NOT bBusy AND NOT bTracking THEN
			nStage := 30;
		END_IF
		
	30:
		fbElevation.Velocity := fElevationMoveVelocity;
		fbElevation.Position := telescopeConfig.elevationHome;
		fbElevation.MoveAxis := TRUE;
		fbAzimuth.Velocity := 10.0;
		fbAzimuth.Position := telescopeConfig.azimuthHome;
		fbAzimuth.MoveAxis := TRUE;
		fbDerotator.Velocity := 10.0;
		fbDerotator.Position := telescopeConfig.derotatorHome;
		fbDerotator.MoveAxis := TRUE;	
		
		IF fbElevation.MoveDone AND 
			fbAzimuth.MoveDone AND 
			fbDerotator.MoveDone THEN
			nStage := 100;
		END_IF
			
	100:
		bPower := FALSE;
		fElevation := fElevationCurrent;
		fAzimuth := fAzimuthCurrent;
		_PowerOn := TRUE;
		bIsParked := FALSE;
		nStage := 0;
	
END_CASE
END_METHOD

METHOD _SendTelemetry : BOOL
VAR_INPUT
END_VAR
SUPER^._PublishTelemetry();

fbComm.Publish('telescope', 'dome', 'TELESCOPE.READY_STATE',	LREAL_TO_STRING(fReadyState));
fbComm.Publish('telescope', 'dome', 'TELESCOPE.MOTION_STATE',	LREAL_TO_STRING(nMotionState));
fbComm.Publish('telescope', 'dome', 'TELESCOPE.INTERRUPTED_AUTO_CLEAR_COUNT', UDINT_TO_STRING(nInterruptedAutoClearCount));

// INFO, CONFIG.MOUNTOPTIONS/MOUNT, STATUS.GLOBAL, OBJECT.INSTRUMENTAL.ALT/AZ and the static
// OBJECT.EQUATORIAL.EPOCH/EQUINOX/RA_PM/DEC_PM/RA_RATE/DEC_RATE fields used to be republished
// here too, byte-identical to what SUPER^._PublishTelemetry() above already sends under the same
// field names from the same source variables -- removed as pure duplication (#22).
//
// OBJECT.EQUATORIAL.RA_ICRS/DEC_ICRS kept even though pybrotlib's schema (the Python MQTT
// consumer, BROTLib/pyBROT src/pybrotlib/telemetry.py) has no such field under
// object.equatorial -- only object.equatorial.ra/dec, which SUPER already publishes with the
// same value -- so this specific publish looks like dead weight for that consumer. Not removing
// it here anyway: Telegraf/InfluxDB ingests the raw MQTT line independent of pybrotlib's schema,
// so something else could still depend on this exact field name landing in Influx. (For contrast,
// POSITION.EQUATORIAL.RA_ICRS/DEC_ICRS -- a different field, published further down -- *is* in
// pybrotlib's schema and is a real, actively consumed field.)
//
// OBJECT.HORIZONTAL.ALT/AZ below is also kept even though SUPER publishes those same field names:
// SUPER's version is conditional on bSlew (fElevation/fAzimuth vs fElevationCalc/fAzimuthCalc);
// this unconditional republish runs after it and is what has actually been on the wire -- changing
// that is a behavior change, not a dedup.

// EQUATORIAL
// all angles in the telemetry are degrees, RA included, like the rightascension command (BROTLib#37)
fbComm.Publish('telescope', 'dome', 'OBJECT.EQUATORIAL.RA_ICRS', LREAL_TO_STRING(fRightAscension));
fbComm.Publish('telescope', 'dome', 'OBJECT.EQUATORIAL.DEC_ICRS', LREAL_TO_STRING(fDeclination));

// HORIZONTAL
fbComm.Publish('telescope', 'dome', 'OBJECT.HORIZONTAL.ALT', LREAL_TO_STRING(fElevationCalc));
fbComm.Publish('telescope', 'dome', 'OBJECT.HORIZONTAL.AZ', LREAL_TO_STRING(fAzimuthCalc));

(* POINTING *)
fbComm.Publish('telescope', 'dome', 'POINTING.SLEWTIME', LREAL_TO_STRING(fSlewtime));
fbComm.Publish('telescope', 'dome', 'POINTING.OFFSETS.ALT', LREAL_TO_STRING(fElevationPointingOffset));
fbComm.Publish('telescope', 'dome', 'POINTING.OFFSETS.AZ', LREAL_TO_STRING(fAzimuthPointingOffset));

(*POSITION*)
//LOCAL
fbComm.Publish('telescope', 'dome', 'POSITION.LOCAL.SIDEREAL_TIME', LREAL_TO_STRING(fLst));
fbComm.Publish('telescope', 'dome', 'POSITION.LOCAL.JD', LREAL_TO_STRING(fJd));
fbComm.Publish('telescope', 'dome', 'POSITION.LOCAL.LATITUDE', LREAL_TO_STRING(telescopeConfig.latitude));
fbComm.Publish('telescope', 'dome', 'POSITION.LOCAL.LONGITUDE', LREAL_TO_STRING(telescopeConfig.longitude));
fbComm.Publish('telescope', 'dome', 'POSITION.LOCAL.HEIGHT', LREAL_TO_STRING(telescopeConfig.altitude));

// INSTRUMENTAL
// > ALT
// POWER_STATE
IF fbElevation.Enable THEN
	fbComm.Publish('telescope', 'dome', 'POSITION.INSTRUMENTAL.ALT.POWER_STATE', '1.0');
ELSE
	fbComm.Publish('telescope', 'dome', 'POSITION.INSTRUMENTAL.ALT.POWER_STATE', '0.0');
END_IF
//REFERENCED
IF fbElevation.Calibrated THEN
	fbComm.Publish('telescope', 'dome', 'POSITION.INSTRUMENTAL.ALT.REFERENCED', '1.0');
ELSE
	fbComm.Publish('telescope', 'dome', 'POSITION.INSTRUMENTAL.ALT.REFERENCED', '0.0');
END_IF
//ERROR_STATE
IF fbElevation.Error THEN
	fbComm.Publish('telescope', 'dome', 'POSITION.INSTRUMENTAL.ALT.ERROR_STATE', UDINT_TO_STRING(fbElevation.ErrorID));
ELSE
	fbComm.Publish('telescope', 'dome', 'POSITION.INSTRUMENTAL.ALT.ERROR_STATE', '0');
END_IF
//MOTION_STATE
IF fbElevation.Busy THEN
	IF fbElevation.isTracking THEN
		fbComm.Publish('telescope', 'dome', 'POSITION.INSTRUMENTAL.ALT.MOTION_STATE', '8');
	ELSE
		fbComm.Publish('telescope', 'dome', 'POSITION.INSTRUMENTAL.ALT.MOTION_STATE', '1');
	END_IF
ELSE
	fbComm.Publish('telescope', 'dome', 'POSITION.INSTRUMENTAL.ALT.MOTION_STATE', '0');
END_IF
fbComm.Publish('telescope', 'dome', 'POSITION.INSTRUMENTAL.ALT.REALPOS', LREAL_TO_STRING(fElevationCurrent-fElevationOffset));
fbComm.Publish('telescope', 'dome', 'POSITION.INSTRUMENTAL.ALT.CURRPOS', LREAL_TO_STRING(fElevationCurrent));
fbComm.Publish('telescope', 'dome', 'POSITION.INSTRUMENTAL.ALT.TARGETPOS', LREAL_TO_STRING(fbElevation.Position));
fbComm.Publish('telescope', 'dome', 'POSITION.INSTRUMENTAL.ALT.CURRSPEED', LREAL_TO_STRING(fbElevation.Velocity));
fbComm.Publish('telescope', 'dome', 'POSITION.INSTRUMENTAL.ALT.TARGETDISTANCE', LREAL_TO_STRING(ABS(fElevationCurrent-fbElevation.Position)));
fbComm.Publish('telescope', 'dome', 'POSITION.INSTRUMENTAL.ALT.OFFSET', LREAL_TO_STRING(fElevationOffset));

// > AZ
// POWER_STATE
IF fbAzimuth.Enable THEN
	fbComm.Publish('telescope', 'dome', 'POSITION.INSTRUMENTAL.AZ.POWER_STATE', '1.0');
ELSE
	fbComm.Publish('telescope', 'dome', 'POSITION.INSTRUMENTAL.AZ.POWER_STATE', '0.0');
END_IF
//REFERENCED
IF fbAzimuth.Calibrated THEN
	fbComm.Publish('telescope', 'dome', 'POSITION.INSTRUMENTAL.AZ.REFERENCED', '1.0');
ELSE
	fbComm.Publish('telescope', 'dome', 'POSITION.INSTRUMENTAL.AZ.REFERENCED', '0.0');
END_IF
//ERROR_STATE
IF fbAzimuth.Error THEN
	fbComm.Publish('telescope', 'dome', 'POSITION.INSTRUMENTAL.AZ.ERROR_STATE', UDINT_TO_STRING(fbAzimuth.ErrorID));
ELSE
	fbComm.Publish('telescope', 'dome', 'POSITION.INSTRUMENTAL.AZ.ERROR_STATE', '0');
END_IF
//MOTION_STATE
IF fbAzimuth.Busy THEN
	IF fbAzimuth.isTracking THEN
		fbComm.Publish('telescope', 'dome', 'POSITION.INSTRUMENTAL.AZ.MOTION_STATE', '8');
	ELSE
		fbComm.Publish('telescope', 'dome', 'POSITION.INSTRUMENTAL.AZ.MOTION_STATE', '1');
	END_IF
ELSE
	fbComm.Publish('telescope', 'dome', 'POSITION.INSTRUMENTAL.AZ.MOTION_STATE', '0');
END_IF

fbComm.Publish('telescope', 'dome', 'POSITION.INSTRUMENTAL.AZ.CURRPOS', LREAL_TO_STRING(fAzimuthCurrent));
fbComm.Publish('telescope', 'dome', 'POSITION.INSTRUMENTAL.AZ.REALPOS', LREAL_TO_STRING(fAzimuthCurrent-F_AzimuthOffsetOnAxis(fAzimuthOffset, fElevationCurrent)));	// M7: was fElevation (stale)
fbComm.Publish('telescope', 'dome', 'POSITION.INSTRUMENTAL.AZ.TARGETPOS', LREAL_TO_STRING(fbAzimuth.Position));
fbComm.Publish('telescope', 'dome', 'POSITION.INSTRUMENTAL.AZ.CURRSPEED', LREAL_TO_STRING(fbAzimuth.Velocity));
fbComm.Publish('telescope', 'dome', 'POSITION.INSTRUMENTAL.AZ.TARGETDISTANCE', LREAL_TO_STRING(ABS(fAzimuthCurrent-fbAzimuth.Position)));
fbComm.Publish('telescope', 'dome', 'POSITION.INSTRUMENTAL.AZ.OFFSET', LREAL_TO_STRING(fAzimuthOffset));


(*HORIZONTAL*)
fbComm.Publish('telescope', 'dome', 'POSITION.HORIZONTAL.ALT', LREAL_TO_STRING(fElevationCurrentSky));
fbComm.Publish('telescope', 'dome', 'POSITION.HORIZONTAL.AZ', LREAL_TO_STRING(fAzimuthCurrentSky));
//fbComm.Publish('telescope', 'dome', 'POSITION.HORIZONTAL.DOME', LREAL_TO_STRING(fbDome.Position));

(*EQUITORIAL*)
fbComm.Publish('telescope', 'dome', 'POSITION.EQUATORIAL.RA_ICRS', LREAL_TO_STRING(fRightAscensionCurrent));	// degrees (BROTLib#37)
fbComm.Publish('telescope', 'dome', 'POSITION.EQUATORIAL.HA_ICRS', LREAL_TO_STRING(fHourAngleCurrent));
fbComm.Publish('telescope', 'dome', 'POSITION.EQUATORIAL.DEC_ICRS', LREAL_TO_STRING(fDeclinationCurrent));
END_METHOD

METHOD PRIVATE _SlewTelescope : USINT
VAR_INPUT
END_VAR
VAR
	SlewEvent:	FB_Eventlog;
	command_timeout: TON;
END_VAR
VAR_STAT
	nStage:		USINT := 0;
	nLastStage:	USINT := 101;
END_VAR
_SlewTelescope := nStage;
command_timeout(IN := nStage < 100, PT := T#600S);
IF command_timeout.Q THEN
	bError := TRUE;
	nErrorID := 16#40;
	bSoftwareError := TRUE;
	nSoftwareErrorID := 16#40;
	bSlew := FALSE;
	nStage := 0;
	RETURN;
END_IF
IF bReset OR bError OR bInterrupted THEN
	nStage := 0;
	RETURN;
END_IF
CASE nStage OF
	0:	
		IF bReady AND bStopped AND NOT bBusy AND NOT bTracking THEN
			nStage := 10;
		END_IF
	10:
		IF fbElevation.Tracking = TRUE OR fbAzimuth.Tracking = TRUE OR fbDerotator.Tracking = TRUE THEN
			fbElevation.Tracking := FALSE;
			fbAzimuth.Tracking := FALSE;
			fbDerotator.Tracking := FALSE;
		ELSE
			nStage := 25;
		END_IF				
	25:
		fbPointing(
			fAzimuth			:= fAzimuth,
			fElevation			:= fElevation,
			fAzimuthOffset		=> fAzimuthPointingOffset,
			fElevationOffset	=> fElevationPointingOffset
		);	
		fbElevation.Position := fElevation + fElevationPointingOffset + fElevationOffset;
		fbElevation.Velocity := fElevationMoveVelocity;
		fbElevation.MoveAxis := TRUE;
		fbAzimuth.Position := fAzimuth + fAzimuthPointingOffset + F_AzimuthOffsetOnAxis(fAzimuthOffset, fElevation);	// M7: was fElevationCalc, mismatched with fAzimuth above
		fbAzimuth.Velocity := 10.0;
		fbAzimuth.MoveAxis := TRUE;
		fbDerotator.Position := fElevation + fDerotatorOffset;
		fbDerotator.Velocity := 10.0;
		fbDerotator.MoveAxis := TRUE;
		IF fbElevation.Busy AND
			fbAzimuth.Busy AND
			fbDerotator.Busy THEN
				nStage := 50;
		END_IF
	50:
		IF fbElevation.MoveDone THEN
			fbElevation.bMoveAxis := FALSE;
		END_IF
		
		IF fbAzimuth.MoveDone THEN
			fbAzimuth.MoveAxis := FALSE;
		END_IF

		IF fbDerotator.MoveDone THEN
			fbDerotator.MoveAxis := FALSE;
		END_IF
		IF NOT bSlewing AND bStopped THEN // all axis standstill
			nStage := 100;
		END_IF
	100:
		fbElevation.MoveAxis := FALSE;
		fbAzimuth.MoveAxis := FALSE;
		fbDerotator.MoveAxis := FALSE;
		fRightAscension := fRightAscensionCalc;
		fDeclination := fDeclinationCalc;
		bSlew := FALSE;
		nStage := 0;
END_CASE
SlewEvent(Trigger := nStage > nLastStage, FormatString := 'Slew progress: %s', OnMessage := USINT_TO_STRING(nStage), Comm := fbComm);
nLastStage := nStage;
END_METHOD

METHOD PRIVATE _StopTelescope : BOOL
VAR_INPUT
END_VAR
IF fbAzimuth.Tracking = TRUE OR fbElevation.Tracking = TRUE OR fbDerotator.Tracking = TRUE THEN
	fbAzimuth.Tracking := FALSE;
	fbElevation.Tracking := FALSE;
	fbDerotator.Tracking := FALSE;
ELSIF fbAzimuth.MoveAxis = TRUE OR  fbElevation.MoveAxis = TRUE OR fbDerotator.MoveAxis = TRUE THEN
	fbAzimuth.MoveAxis := FALSE;
	fbElevation.MoveAxis := FALSE;
	fbDerotator.MoveAxis := FALSE;
ELSE
	// Only issue Axis stop commands if they are moving
	IF NOT fbAzimuth.fbAxis.StandStill THEN
		fbAzimuth.StopAxis := TRUE;
	ELSE
		fbAzimuth.StopAxis := FALSE;
	END_IF
	
	IF NOT fbElevation.fbAxis.StandStill THEN
		fbElevation.StopAxis := TRUE;
	ELSE
		fbElevation.StopAxis := FALSE;
	END_IF	
	
	IF NOT fbDerotator.fbAxis.StandStill THEN
		fbDerotator.StopAxis := TRUE;
	ELSE
		fbDerotator.StopAxis := FALSE;
	END_IF	

	IF bStopped THEN
		fbAzimuth.StopAxis := FALSE;
		fbElevation.StopAxis := FALSE;
		fbDerotator.StopAxis := FALSE;
		_StopTelescope := FALSE;
	END_IF
END_IF
END_METHOD

METHOD PRIVATE _TrackTelescope : BOOL
VAR_INPUT
END_VAR
// Elevation
fDerotatorVelocity := F_Derotatorvelocity(fAzimuthCalc, fElevationCalc, telescopeConfig.latitude, fDerotatorSign);
fElevationVelocity := F_Elevationvelocity(fAzimuthCalc, telescopeConfig.latitude);
fAzimuthVelocity := F_Azimuthvelocity(fElevationCalc, fAzimuthCalc, telescopeConfig.latitude);
IF fElevationCurrent < 5.0 OR fElevationCurrent > 89.5 THEN
	bTrack := FALSE;
END_IF
IF fAzimuthCurrent > 440.0 THEN
	bTrack := FALSE;
END_IF
IF (fDerotatorCurrent < -69.0 AND fDerotatorVelocity<0.0) OR (fDerotatorCurrent > 379.0 AND fDerotatorVelocity>0.0) THEN
	bTrack := FALSE;
END_IF

fbElevation.Position := fElevationCalc;
IF NOT fbElevation.Tracking THEN
	fbElevation.Velocity := fElevationMoveVelocity;
	fbElevation.MoveAxis := TRUE;
	IF NOT fbElevation.Busy AND fbElevation.MoveDone THEN
		fbElevation.MoveAxis := FALSE;
		IF fbElevation.isTracking THEN
			fbElevation.Velocity := fElevationVelocity;
		ELSE
			fbElevation.Velocity := 3.0*fElevationVelocity;
		END_IF
		fbElevation.Velocity := fElevationVelocity;
		fbElevation.Tracking := TRUE;
	END_IF
ELSE
	fbElevation.Velocity := fElevationVelocity;
END_IF

// Azimuth
fbAzimuth.Position := fAzimuthCalc;
IF NOT fbAzimuth.Tracking THEN
	fbAzimuth.Velocity := 10.0;
	fbAzimuth.MoveAxis := TRUE;
	IF NOT fbAzimuth.Busy AND fbAzimuth.MoveDone THEN
		fbAzimuth.MoveAxis := FALSE;
		IF fbAzimuth.isTracking THEN
			fbAzimuth.Velocity := fAzimuthVelocity;
		ELSE
			fbAzimuth.Velocity := 3.0*fAzimuthVelocity;
		END_IF
		fbAzimuth.Velocity := fAzimuthVelocity;
		fbAzimuth.Tracking := TRUE;
	END_IF
ELSE
	fbAzimuth.Velocity := fAzimuthVelocity;
END_IF

// Derotator
fbDerotator.Position := fDerotatorCalc;
IF NOT fbDerotator.Tracking THEN
	fbDerotator.Velocity := 10.0;
	fbDerotator.MoveAxis := TRUE;
	IF NOT fbDerotator.Busy AND fbDerotator.MoveDone THEN
		fbDerotator.MoveAxis := FALSE;
		IF fbDerotator.isTracking THEN
			fbDerotator.Velocity := fDerotatorVelocity;
		ELSE
			fbDerotator.Velocity := 3.0*fDerotatorVelocity;
		END_IF
		fbDerotator.Velocity := fDerotatorVelocity;
		fbDerotator.Tracking := TRUE;
	END_IF
ELSE
	fbDerotator.Velocity := fDerotatorVelocity;
END_IF
END_METHOD

PROPERTY Altitude : LREAL
GET
Altitude := THIS^.fElevationCurrent;
END_GET
END_PROPERTY

PROPERTY Azimuth : LREAL
GET
Azimuth := THIS^.fAzimuthCurrent;
END_GET
END_PROPERTY

PROPERTY CoverAutoOpen : BOOL
GET
CoverAutoOpen := THIS^.bCoverAutoOpen;
END_GET
SET
// This property has no effect on MONET: _PowerOn always opens the covers
// unconditionally and never reads bCoverAutoOpen. Forcing it TRUE here keeps
// the property honest, but does not by itself guarantee the invariant, since
// bCoverAutoOpen is a public VAR_INPUT a caller can still write to directly.
THIS^.bCoverAutoOpen := TRUE;
END_SET
END_PROPERTY

PROPERTY Declination : LREAL
GET
Declination := THIS^.fDeclination;
END_GET
END_PROPERTY

METHOD Init : BOOL
bPower := TRUE;
END_METHOD

METHOD MoveAltAz : BOOL
VAR_INPUT
	AltAz	: BROTLib.ST_AltAzCoordinate;
END_VAR
fElevation 	:= AltAz.Altitude;
fAzimuth 	:= AltAz.Azimuth;
bSlew		:= TRUE;
END_METHOD

METHOD MoveRaDec : BOOL
VAR_INPUT
	RaDec	: BROTLib.ST_RaDecCoordinate;
END_VAR
fRightAscension	:= RaDec.RightAscension;
fDeclination	:= RaDec.Declination;
bGoto			:= TRUE;
END_METHOD

METHOD Park : BOOL
bPark := TRUE;
END_METHOD

METHOD Reset : BOOL
bReset := TRUE;
END_METHOD

PROPERTY RightAscension : LREAL
GET
RightAscension := THIS^.fRightAscension;
END_GET
END_PROPERTY

METHOD SetAltitudeOffset : BOOL
VAR_INPUT
	Offset	: LREAL;
END_VAR
fElevationOffset := Offset;
END_METHOD

METHOD SetAzimuthOffset : BOOL
VAR_INPUT
	Offset	: LREAL;
END_VAR
fAzimuthOffset := Offset;
END_METHOD

METHOD SetDerotatorOffset : BOOL
VAR_INPUT
	Offset	: LREAL;
END_VAR
fDerotatorOffset := Offset;
END_METHOD

METHOD Slew : BOOL
VAR_INPUT
	fAzimuth	: LREAL;
	fAltitude	: LREAL;
END_VAR
THIS^.fElevation 	:= fAltitude;
THIS^.fAzimuth 	:= fAzimuth;
THIS^.bSlew		:= TRUE;
END_METHOD

METHOD Stop : BOOL
bStop := TRUE;
END_METHOD

METHOD Track : BOOL
VAR_INPUT
	fRightAscension	: LREAL;
	fDeclination	: LREAL;
END_VAR
THIS^.fRightAscension	:= fRightAscension;
THIS^.fDeclination		:= fDeclination;
//THIS^.bTrack			:= TRUE;
THIS^.bGoto				:= TRUE;
END_METHOD

METHOD TrackRaDec : BOOL
VAR_INPUT
	RaDec	: BROTLib.ST_RaDecCoordinate;
END_VAR
fRightAscension	:= RaDec.RightAscension;
fDeclination		:= RaDec.Declination;
//bTrack			:= TRUE;
THIS^.bGoto				:= TRUE;
END_METHOD

END_FUNCTION_BLOCK

// ---- F_AzimuthOffsetOnAxis.TcPOU
// Azimuth-axis correction (degrees) for a cross-elevation offset on the sky (fAzimuthOffset, degrees) at
// elevation fElevation (degrees): fAzimuthOffset / COS(fElevation). Near the zenith 1/COS grows without bound and
// is a division by zero at 90 deg, so COS is floored at COS(89.5 deg) (factor 115 at most) and the result is limited
// to +-10 deg, the same bound BROTLib puts on the offset command (BROTLib#27). Below 89.5 deg the result is unchanged.
FUNCTION F_AzimuthOffsetOnAxis : LREAL
VAR_INPUT
	fAzimuthOffset	: LREAL;	// cross-elevation offset on the sky, degrees
	fElevation		: LREAL;	// elevation, degrees
END_VAR
VAR CONSTANT
	D2R				: LREAL := 0.017453292519943295;
	MIN_COS			: LREAL := 0.008726535498373935;	// COS(89.5 deg)
	MAX_AXIS_OFFSET	: LREAL := 10.0;					// degrees
END_VAR

F_AzimuthOffsetOnAxis := LIMIT(-MAX_AXIS_OFFSET, fAzimuthOffset / MAX(COS(fElevation * D2R), MIN_COS), MAX_AXIS_OFFSET);

END_FUNCTION

// ---- FB_MonetSafetyHandling.TcPOU
FUNCTION_BLOCK FB_MonetSafetyHandling
VAR
	// power on delay

	// AT%I*/AT%Q* below are mapped directly on this FB: only one instance per PLC is
	// supported, a second instance would collide on the same physical hardware.
	inError					AT%I*:	BOOL;		// Safety Error Condition
	outRun					AT%Q*:	BOOL;		// Run/Stop Safety
	outRestart				AT%Q*:	BOOL;		// Restart Safety
	outErrAck				AT%Q*:	BOOL;		// Error Acknowledgement 
	
	outResetAzimuthSTO		AT%Q*: BOOL;
	outResetElevationSTO	AT%Q*: BOOL;
	outResetDerotatorSTO	AT%Q*: BOOL;
	
	// Safety group
	fbInfoGroup1			: FB_InfoGroup;
	stInfoGroup1	AT%I*	: ST_InfoDataGroup;
	sStateGroup1			: STRING;
	
	// Estop
	fbInfoEStop1			:FB_InfoEStop;
	stInfoEStop1 	AT%I*	:ST_InfoDataFB;
	sStateEStop1			:STRING;
	sDiagEStop1				:STRING;	
	
	// Info EL1904
	fbInfoSafetyIn			: FB_InfoConnection;
	stInfoSafetyIn 	AT%I*	: ST_InfoDataConnection;
	sStateSafetyIn			: STRING;
	sDiagSafetyIn			: STRING;
	bSafetyInCh1			: BOOL;
	bSafetyInCh2			: BOOL;
	bSafetyInCh3			: BOOL;
	bSafetyInCh4			: BOOL;
	
	// Info EL2904
	fbInfoSafetyOut			: FB_InfoConnection;
	stInfoSafetyOut AT%I*	: ST_InfoDataConnection;
	sStateSafetyOut			: STRING;
	sDiagSafetyOut			: STRING;
	bSafetyOutCh1			: BOOL;
	bSafetyOutCh2			: BOOL;
	bSafetyOutCh3			: BOOL;
	bSafetyOutCh4			: BOOL;
	
	initialStartUpStep		: INT := 0;
	startDelay 				: TON := (PT := T#2S);
	stateDelay 				: TON := (PT := T#1S);

	// external reset request (cabinet/pendant reset button)
	rtrigReset				: R_TRIG;
	resetStep				: INT := 0;
	resetDelay				: TON := (PT := T#1S);

	ErrAckLog				: FB_EventLog;		// Errack logging
	RestartLog				: FB_EventLog;		// restart logging
	SafetyLog				: FB_EventLog;		// safety logging

	fbComm					: I_Comm;
END_VAR
VAR_OUTPUT
	error					: BOOL;		// error condition
	state          			: BOOL;		// safety is okay
	estop					: BOOL;		// Emergency_stop engaged
END_VAR
VAR_INPUT
	// issue a remote restart
	//remote_restart:		BOOL;
	// issue a remute run/stop
	remote_run		: BOOL := TRUE;
	// cabinet/pendant reset button: toggles Restart, then ErrAck
	resetRequest	: BOOL;
END_VAR

// Safety is running on start
outRun := remote_run;

// error?
error := inError;

// get safety status
fbInfoGroup1(
	stInfoData	:= stInfoGroup1,
	sState		=> sStateGroup1);
state := sStateGroup1 = 'RUN' OR initialStartUpStep <> 100;

// estop triggered?
fbInfoEStop1(
	stInfoData	:= stInfoEStop1, 
	sState		=> sStateEStop1, 
	sDiag		=> sDiagEStop1);
estop := sStateEStop1 <> 'RUN' AND initialStartUpStep = 100;

//Info SafetyIn EL1904
fbInfoSafetyIn(
	stInfoData		:=stInfoSafetyIn, 
	sState			=>sStateSafetyIn, 
	sDiag			=>sDiagSafetyIn, 
	bChannel1		=>bSafetyInCh1, 
	bChannel2		=>bSafetyInCh2, 
	bChannel3		=>bSafetyInCh3, 
	bChannel4		=>bSafetyInCh4);	
	
//Info SafetyOut EL2904
fbInfoSafetyOut(
	stInfoData		:=stInfoSafetyOut, 
	sState			=>sStateSafetyOut, 
	sDiag			=>sDiagSafetyOut, 
	bChannel1		=>bSafetyOutCh1, 
	bChannel2		=>bSafetyOutCh2, 
	bChannel3		=>bSafetyOutCh3, 
	bChannel4		=>bSafetyOutCh4);
	
// initial startup	
CASE initialStartUpStep OF
	0:
		// begin start up procedure, do ErrAck
		startDelay(IN := TRUE);
		IF startDelay.Q THEN
			startDelay(IN := FALSE);
			initialStartUpStep := 10;
		END_IF		
	10:
		// do err ack 
		outErrAck := TRUE;
		stateDelay(IN := TRUE);
		IF stateDelay.Q THEN
			stateDelay(IN := FALSE);
			outErrAck := FALSE;
			initialStartUpStep := 20;
		END_IF
	20:
		// do restart
		outRestart := TRUE;
		stateDelay(IN := TRUE);
		IF stateDelay.Q THEN
			stateDelay(IN := FALSE);
			outRestart := FALSE;
			initialStartUpStep := 30;
		END_IF		
	30:
		// do STO restart
		outResetAzimuthSTO := TRUE;
		outResetElevationSTO := TRUE;
		outResetDerotatorSTO := TRUE;
		stateDelay(IN := TRUE);
		IF stateDelay.Q THEN
			stateDelay(IN := FALSE);
			outResetAzimuthSTO := FALSE;
			outResetElevationSTO := FALSE;
			outResetDerotatorSTO := FALSE;
			initialStartUpStep := 100;
		END_IF			
END_CASE

// external reset request (cabinet/pendant button): toggle Restart, then ErrAck
rtrigReset(CLK := resetRequest);
IF rtrigReset.Q THEN
	resetStep := 10;
END_IF

CASE resetStep OF
	10:
		outRestart := TRUE;
		resetDelay(IN := TRUE);
		IF resetDelay.Q THEN
			resetDelay(IN := FALSE);
			outRestart := FALSE;
			resetStep := 20;
		END_IF
	20:
		outErrAck := TRUE;
		resetDelay(IN := TRUE);
		IF resetDelay.Q THEN
			resetDelay(IN := FALSE);
			outErrAck := FALSE;
			resetStep := 0;
		END_IF
END_CASE


ErrAckLog(
	Trigger 	:= outErrAck,
	OnMessage 	:= 'Safety error was acknowledged.',
	Comm		:= fbComm
);
			
RestartLog(	
	Trigger 	:= outRestart,
	Level 		:= ADSLOG_MSGTYPE_WARN,
	OnMessage 	:= 'Safety was restarted.',
	Comm		:= fbComm
);

SafetyLog(	
	Trigger 	:= estop,
	Level 		:= ADSLOG_MSGTYPE_ERROR,
	OnMessage 	:= 'Safety Error! Emergency stop engaged!',
	OffMessage 	:= 'Safety is OK.',
	OffLevel 	:= ADSLOG_MSGTYPE_HINT,
	Comm		:= fbComm);

//FB_Init is always available implicitly and it is used primarily for initialization.
//The return value is not evaluated. For a specific influence, you can also declare the
//methods explicitly and provide additional code there with the standard initialization
//code. You can evaluate the return value.
METHOD FB_Init: BOOL
VAR_INPUT
    bInitRetains	: BOOL; // TRUE: the retain variables are initialized (reset warm / reset cold)
    bInCopyCode		: BOOL;  // TRUE: the instance will be copied to the copy code afterward (online change)
	comm			: I_Comm;	      
END_VAR
THIS^.fbComm := comm;
END_METHOD

END_FUNCTION_BLOCK

// ---- FB_MonetMqttWatchdog.TcPOU
// Safe state when the MQTT broker is gone: after tGrace without a connection, park the telescope and close the
// roof, since nobody (pyobs, weather/roof logic on the observatory computer) can command or protect it any more.
// Armed only after the first successful connect, so a slow or normal boot never trips it. Moved unchanged from
// MONETS's MAIN so that MONET/S and MONET/N share it.
FUNCTION_BLOCK FB_MonetMqttWatchdog
VAR_INPUT
	bConnected		: BOOL;				// fbComm.bConnected
	iTelescope		: I_Telescope;		// parked on timeout
	iRoof			: I_Roof;			// closed on timeout
	tGrace			: TIME := T#30S;	// grace period before the emergency shutdown
END_VAR
VAR_OUTPUT
	bTriggered		: BOOL;				// TRUE while the watchdog holds the telescope parked and the roof closed
END_VAR
VAR
	fbComm			: I_Comm;
	tonWatchdog		: TON;
	bEverConnected	: BOOL := FALSE;
END_VAR

bEverConnected := bEverConnected OR bConnected;
tonWatchdog(IN := bEverConnected AND NOT bConnected, PT := tGrace);
bTriggered := tonWatchdog.Q;

IF bTriggered THEN
	IF iTelescope <> 0 THEN
		iTelescope.Park();
	END_IF
	IF iRoof <> 0 THEN
		iRoof.Close();
	END_IF
	fbComm.Publish('electronics', 'base', 'MQTTWatchdog', 'TRIGGERED');
END_IF

METHOD FB_Init: BOOL
VAR_INPUT
    bInitRetains	: BOOL; // TRUE: the retain variables are initialized (reset warm / reset cold)
    bInCopyCode		: BOOL;  // TRUE: the instance will be copied to the copy code afterward (online change)
	comm			: I_Comm;
END_VAR
THIS^.fbComm := comm;
END_METHOD

END_FUNCTION_BLOCK

// ---- FB_MonetPendantControl.TcPOU
FUNCTION_BLOCK FB_MonetPendantControl
VAR_INPUT
	eTelescopeMode		: E_TelescopeMode;
	fbCovers			: REFERENCE TO FB_MonetCoverControl;
	fbBrake				: REFERENCE TO FB_HydraulicsControl;
	fbHydraulics		: REFERENCE TO FB_HydraulicsControl;
	fbFocus		 		: REFERENCE TO FB_FocusControl;
	fbElevation			: REFERENCE TO FB_ElevationControl;
	fbAzimuth	 		: REFERENCE TO FB_AzimuthControl;
	fbDerotator			: REFERENCE TO FB_DerotatorControl;
END_VAR
VAR_OUTPUT
	bEnable				: BOOL;
END_VAR
VAR
	fbComm				: I_Comm;
	nSelection			: UINT;		// program selection of the pendant control
	bError				: BOOL;		// error on the pendant control
	bHorn				: BOOL;
	fbStartTrigger		: R_TRIG;
	fbUpTrigger			: R_TRIG;
	fbDownTrigger		: R_TRIG;	
	fbResetTrigger		: R_TRIG;

	//DIN17 2.0
	// AT%I*/AT%Q* below are mapped directly on this FB: only one instance per PLC is
	// supported, a second instance would collide on the same physical hardware.
	IbBCD0				AT%I*: BOOL;
	IbBCD2				AT%I*: BOOL;
	IbBCD4				AT%I*: BOOL;
	IbBCD8				AT%I*: BOOL;
	IbResetButton		AT%I*: BOOL;
	IbDirectionUp		AT%I*: BOOL;
	IbDirectionDown		AT%I*: BOOL;
	IbEnableKey			AT%I*: BOOL;
	IbEnableButton		AT%I*: BOOL;
	IbDirectionLeft		AT%I*: BOOL;
	IbDirectionRight	AT%I*: BOOL;

	ObLampUp			AT%Q*: BOOL;
	ObLampDown			AT%Q*: BOOL;
	ObLampRight			AT%Q*: BOOL;
	ObLampLeft			AT%Q*: BOOL;
	ObLampError			AT%Q*: BOOL;	
END_VAR

(* 
This program is responsible for the manual control of the telescope.
all movable parts can be controlled from here. This is mainly for testing and
maintenance.
WARNING! Some of the safety routines are disabled, when operating the telescope manually.
*)
// calculate the value of the selector
nSelection := 1*BOOL_TO_UINT(IbBCD0) + 
			 2*BOOL_TO_UINT(IbBCD2) + 
			 4*BOOL_TO_UINT(IbBCD4) +
			 8*BOOL_TO_UINT(IbBCD8);

// detect disconnection of the manual controls (should also trigger emergency stop).			 
bError := (nSelection = 0);

// disable all the lamps
ObLampLeft := FALSE;
ObLampRight := FALSE;
ObLampUp := FALSE;
ObLampDown := FALSE;
bHorn := FALSE;

fbUpTrigger(CLK := IbDirectionUp);
fbDownTrigger(CLK := IbDirectionDown);
//R_Enable(CLK := enable);
// the error lamp is the same as the error lamp of the main panel
ObLampError := ObLampError;

// enabled?
bEnable := IbEnableKey;
IF NOT bEnable THEN
	RETURN;
END_IF

// reset or start pushed?
fbResetTrigger(CLK := IbResetButton);
fbStartTrigger(CLK := IbEnableButton);

// mode
IF eTelescopeMode = E_TelescopeMode.automatic THEN
	;
END_IF

// enable only the selected item and connect lamps and buttons accordingly
CASE nSelection OF
	1, 2, 3:	// reserved for Cover 1-3 control
		ObLampUp := fbCovers.Opened;
		ObLampDown := fbCovers.Closed;
		IF IbEnableKey THEN
			fbCovers.bOpen := IbDirectionUp AND fbCovers.Opened;
			fbCovers.bClose := IbDirectionDown AND fbCovers.Closed;
			ObLampError := fbCovers.bError;	
		ELSE
			IF IbDirectionDown THEN 
				fbCovers.Close();
			ELSIF IbDirectionUp THEN
				fbCovers.Open();
			END_IF		
		END_IF
		
	4:	// Nasmyth / mirror M3 control
		
	5:	// Focus Control
		IF __ISVALIDREF(fbFocus) THEN
			fbFocus.Enable := IbEnableButton;			
			ObLampUp := fbFocus.Enable AND fbFocus.Ready AND NOT fbFocus.InPosLimit;
			ObLampDown := fbFocus.Enable AND fbFocus.Ready AND NOT fbFocus.InNegLimit;
			fbFocus.MovePos := IbDirectionUp;
			fbFocus.MoveNeg := IbDirectionDown;
			IF fbResetTrigger.Q THEN
				fbFocus.Reset();
			END_IF
			ObLampError := fbFocus.Error;
		END_IF
							
	6:	// Derotator control
		fbDerotator.Enable := IbEnableButton;
		ObLampLeft  := fbDerotator.Ready AND NOT fbDerotator.InNegLimit;
		ObLampRight := fbDerotator.Ready AND NOT fbDerotator.InPosLimit;
		fbDerotator.MoveNeg := IbDirectionLeft AND NOT fbDerotator.inDigitalInputs.1;
		fbDerotator.MovePos := IbDirectionRight AND NOT fbDerotator.inDigitalInputs.0;
		ObLampError := fbDerotator.Error;
		IF fbResetTrigger.Q THEN
			fbDerotator.Reset();
		END_IF
		
							
	7:	// Elevation Control
		fbElevation.Enable := IbEnableButton;		
		fbElevation.MovePos := IbDirectionUp AND fbElevation.inDigitalInputs.0;
		fbElevation.MoveNeg := IbDirectionDown AND fbElevation.inDigitalInputs.1;
		ObLampUp := fbElevation.inDigitalInputs.0;
		ObLampDown := fbElevation.inDigitalInputs.1;
		ObLampError := fbElevation.bError;
		IF fbResetTrigger.Q THEN
			fbElevation.Reset();
		END_IF
		
	8:	// Azimuth Control
		fbAzimuth.Enable := IbEnableButton;
		ObLampLeft := fbAzimuth.inDigitalInputs.0; // NOT GVL_Telescope.azimut_limit_switch;
		ObLampRight := fbAzimuth.inDigitalInputs.1; // NOT GVL_Telescope.azimut_limit_switch;
		fbAzimuth.MoveNeg := IbDirectionLeft AND fbAzimuth.inDigitalInputs.0;
		fbAzimuth.MovePos := IbDirectionRight AND fbAzimuth.inDigitalInputs.1;
		IF fbResetTrigger.Q THEN
			fbAzimuth.Reset();
		END_IF

END_CASE

//FB_Init is always available implicitly and it is used primarily for initialization.
//The return value is not evaluated. For a specific influence, you can also declare the
//methods explicitly and provide additional code there with the standard initialization
//code. You can evaluate the return value.
METHOD FB_Init: BOOL
VAR_INPUT
    bInitRetains: BOOL; // TRUE: the retain variables are initialized (reset warm / reset cold)
    bInCopyCode: BOOL;  // TRUE: the instance will be copied to the copy code afterward (online change)
	comm			: I_Comm;   
END_VAR
THIS^.fbComm 	:= comm;
END_METHOD

END_FUNCTION_BLOCK

// ---- FB_MonetPowerMonitoring.TcPOU
FUNCTION_BLOCK FB_MonetPowerMonitoring
VAR_INPUT
END_VAR
VAR_OUTPUT
	phaseOK:				BOOL;
END_VAR
VAR
	fbComm					: I_Comm;	

	// AT%I*/AT%Q* below are mapped directly on this FB: only one instance per PLC is
	// supported, a second instance would collide on the same physical hardware.
	FrequencyGuardWarning	AT%I*: BOOL;
	FrequencyGuardError		AT%I*: BOOL;
	QualityGuardWarning		AT%I*: BOOL;
	QualityGuardError		AT%I*: BOOL;
	UnbalanceGuardWarning	AT%I*: BOOL;
	UnbalanceGuardError		AT%I*: BOOL;
	PowerQuality			AT%I*: REAL;
	L1OverVoltage			AT%I*: BOOL;
	L1InaccVoltage			AT%I*: BOOL;
	L1VoltageGuardWarning	AT%I*: BOOL;
	L1VoltageGuardError		AT%I*: BOOL;
	L2OverVoltage			AT%I*: BOOL;
	L2InaccVoltage			AT%I*: BOOL;
	L2VoltageGuardWarning	AT%I*: BOOL;
	L2VoltageGuardError		AT%I*: BOOL;
	L3OverVoltage			AT%I*: BOOL;
	L3InaccVoltage			AT%I*: BOOL;
	L3VoltageGuardWarning	AT%I*: BOOL;
	L3VoltageGuardError		AT%I*: BOOL;
	
	mqttTimer: 				TON := (PT:=T#10S);
	powerWarningDelay:		TON := (PT:=T#100MS);
	powerWarningRetain:		TOF := (PT:=T#2000MS);
	
	powerError:				FB_EventLog;
	powerWarning:			FB_EventLog;
END_VAR

// M5: previously ignored *GuardError entirely (only PowerError's log message used them)
// and QualityGuard*/UnbalanceGuard* altogether; phaseOK now gates bMainReady (see MONETcommon#11).
phaseOK := NOT FrequencyGuardWarning AND NOT FrequencyGuardError AND
	NOT QualityGuardWarning AND NOT QualityGuardError AND
	NOT UnbalanceGuardWarning AND NOT UnbalanceGuardError AND
	NOT L1VoltageGuardWarning AND NOT L1VoltageGuardError AND
	NOT L2VoltageGuardWarning AND NOT L2VoltageGuardError AND
	NOT L3VoltageGuardWarning AND NOT L3VoltageGuardError;

powerWarningDelay(IN := NOT phaseOK);
powerWarningRetain(IN := powerWarningDelay.Q);

// MQTT Section
mqttTimer(IN:=TRUE);
IF mqttTimer.Q THEN
	mqttTimer(IN:=FALSE);

	fbComm.Publish('power', 'power', 'FrequencyGuardWarning',	BOOL_TO_STRING(FrequencyGuardWarning));
	fbComm.Publish('power', 'power', 'FrequencyGuardError',	BOOL_TO_STRING(FrequencyGuardError));
	fbComm.Publish('power', 'power', 'QualityGuardWarning',	BOOL_TO_STRING(QualityGuardWarning));
	fbComm.Publish('power', 'power', 'QualityGuardError',		BOOL_TO_STRING(QualityGuardError));
	fbComm.Publish('power', 'power', 'UnbalanceGuardWarning',	BOOL_TO_STRING(UnbalanceGuardWarning));
	fbComm.Publish('power', 'power', 'UnbalanceGuardError',	BOOL_TO_STRING(UnbalanceGuardError));
	fbComm.Publish('power', 'power', 'PowerQuality',			REAL_TO_STRING(PowerQuality));
	fbComm.Publish('power', 'power', 'L1OverVoltage',			BOOL_TO_STRING(L1OverVoltage));
	fbComm.Publish('power', 'power', 'L1InaccVoltage',		BOOL_TO_STRING(L1InaccVoltage));
	fbComm.Publish('power', 'power', 'L1VoltageGuardWarning',	BOOL_TO_STRING(L1VoltageGuardWarning));
	fbComm.Publish('power', 'power', 'L1VoltageGuardError',	BOOL_TO_STRING(L1VoltageGuardError));
	fbComm.Publish('power', 'power', 'L2OverVoltage',			BOOL_TO_STRING(L2OverVoltage));
	fbComm.Publish('power', 'power', 'L2InaccVoltage',		BOOL_TO_STRING(L2InaccVoltage));
	fbComm.Publish('power', 'power', 'L2VoltageGuardWarning',	BOOL_TO_STRING(L2VoltageGuardWarning));
	fbComm.Publish('power', 'power', 'L2VoltageGuardError',	BOOL_TO_STRING(L2VoltageGuardError));
	fbComm.Publish('power', 'power', 'L3OverVoltage',			BOOL_TO_STRING(L3OverVoltage));
	fbComm.Publish('power', 'power', 'L3InaccVoltage',		BOOL_TO_STRING(L3InaccVoltage));
	fbComm.Publish('power', 'power', 'L3VoltageGuardWarning',	BOOL_TO_STRING(L3VoltageGuardWarning));
	fbComm.Publish('power', 'power', 'L3VoltageGuardError',	BOOL_TO_STRING(L3VoltageGuardError));
END_IF

// EventLog section
PowerError(	
	Trigger 		:= FrequencyGuardError OR QualityGuardError OR UnbalanceGuardError OR L1VoltageGuardError OR L2VoltageGuardError OR L3VoltageGuardError, 
	Level 			:= ADSLOG_MSGTYPE_ERROR,
	FormatString 	:= '%s',
	OnMessage 		:= 'electrical power:	ERROR!',
	comm			:= fbComm);
	
PowerWarning(	
	Trigger 		:= powerWarningRetain.Q, 
	Level 			:= ADSLOG_MSGTYPE_WARN,
	FormatString 	:= '%s',
	OnMessage 		:= 'electrical power:	WARNING!',
	comm			:= fbComm);

//FB_Init is always available implicitly and it is used primarily for initialization.
//The return value is not evaluated. For a specific influence, you can also declare the
//methods explicitly and provide additional code there with the standard initialization
//code. You can evaluate the return value.
METHOD FB_Init: BOOL
VAR_INPUT
    bInitRetains	: BOOL; // TRUE: the retain variables are initialized (reset warm / reset cold)
    bInCopyCode		: BOOL;  // TRUE: the instance will be copied to the copy code afterward (online change)
	comm			: I_Comm;	   
END_VAR
THIS^.fbComm := comm;
END_METHOD

END_FUNCTION_BLOCK
